# B&R Automation Studio project 8238 (part 21)

#### mnTestCyclic.st - Cyclic code
```iecst
(********************************************************************
 * COPYRIGHT -- Herbert Kannegiesser GmbH
 ********************************************************************
 * Program: mnTest
 * File: mnTestCyclic.st
 * Author: hunholz
 * Created: March 03, 2012
 ********************************************************************
 * Implementation of program mnTest
 ********************************************************************)

PROGRAM _CYCLIC

	//====================
	// Kommandointerpreter
	//====================

	CASE _CommandoState OF

		_csIdle:

			CASE mnTestCmd.Request.Command.wCommand OF

				KG_CMD_NOCOMMAND:

					mnTestCmd.Response.wCmdStatus := KG_CMD_NOCOMMAND;

				MNTEST_CMD_RESET:

					IF mnTestCmd.Request.Command.lData0 <> MNTEST_RESETMODE_WARMSTART AND mnTestCmd.Request.Command.lData0 <> MNTEST_RESETMODE_COLDSTART THEN

						mnTestCmd.Response.wCmdStatus := KG_CMDSTAT_INVALID_PARAMETER;

					ELSE

						SYSreset(enable := TRUE, mode := UDINT_TO_USINT(mnTestCmd.Request.Command.lData0));
						mnTestCmd.Response.wCmdStatus := MNTEST_CMD_RESET;

					END_IF

					_CommandoState := _csWaitForNull;

				MNTEST_CMD_SETMODE:

					IF _wTestMode <> 0 THEN

						mnTestCmd.Response.wCmdStatus := MNTEST_CMDSTAT_SETMODEFAILED;

					ELSIF mnTestCmd.Request.Command.lData0 = 0 OR mnTestCmd.Request.Command.lData0 > MNTEST_TESTMODE_MAX THEN

						mnTestCmd.Response.wCmdStatus := KG_CMDSTAT_INVALID_PARAMETER;

					ELSE

						IF IFmnParam.Out.xParamOK THEN
							_wTestMode := UDINT_TO_UINT(mnTestCmd.Request.Command.lData0);
							mnTestCmd.Response.wCmdStatus := MNTEST_CMD_SETMODE;
							_TestState := _tsSetMode;
						END_IF

					END_IF

					_CommandoState := _csWaitForNull;

				ELSE

					_CommandoState := _csWaitForNull;
					mnTestCmd.Response.wCmdStatus := KG_CMDSTAT_NOTVALID;

			END_CASE

		_csWaitForNull:

			IF mnTestCmd.Request.Command.wCommand = KG_CMD_NOCOMMAND THEN

				_CommandoState := _csIdle;
				mnTestCmd.Response.wCmdStatus := KG_CMD_NOCOMMAND;

			END_IF

		ELSE

			_CommandoState := _csIdle;

	END_CASE

	//======================
	// Statemachine Testmode
	//======================

	CASE _TestState OF

		_tsIdle:

			// Tue nichts

		_tsSetMode:

			_sMachineNo := WSTRING_TO_STRING(IFmnParam.Out.utfMachineNumber);

			_fbSetMode(enable := TRUE, pStruc := IFmnTest.In.pStrucTest, wMode := _wTestMode, sMachineNo := _sMachineNo);

			IF _fbSetMode.status = ERR_OK THEN

				IF _wTestMode = 1 THEN

					// Framework darf keine Meldungen mehr erzeugen und das
					// Meldesystem wird zurückgesetzt
					IFmnTest.Out.xNoMessages := TRUE;
					brsmemset(ADR(kgMsgStatus),0,SIZEOF(kgMsgStatus));

					_TestState := _tsPrepTest1;

				ELSIF _wTestMode = 2 THEN

					brsmemset(ADR(kgMsgStatus),0,SIZEOF(kgMsgStatus));

					_TestState := _tsRun;

				END_IF

			ELSE

				_TestState := _tsFault;

				mnTestStat.wStatus := MNTEST_STAT_ERRFBSETMODE;
				mnTestStat.sStatus := UINT_TO_STRING(_fbSetMode.status);

			END_IF

		_tsPrepTest1:

			_doInfoCfg.enable := TRUE;	// VAR_INPUT BOOL enable 'enables execution'
			_doInfoCfg.pName := ADR('CfgMsgStat');	// VAR_INPUT UDINT pName 'name of data object'
			_doInfoCfg();

			IF _doInfoCfg.status = ERR_OK THEN

				_wMsgCnt := UDINT_TO_UINT((_doInfoCfg.len-SIZEOF(UINT))/SIZEOF (MsgCfgLine_Typ)); // Laenge der Version zu Beginn abziehen

				IF _wMsgCnt > 0 AND _wMsgCnt <= MNMSG_MAX_CFGMESSAGES THEN

					_MsgCfgList ACCESS _doInfoCfg.pDatObjMem + SIZEOF(UINT);
					_TestState := _tsRun;

				ELSE
					// Meldungskonfiguration fehlerhaft
					_TestState := _tsFault;

					mnTestStat.wStatus := MNTEST_STAT_ERRMSGCFGCNT;
					mnTestStat.sStatus := UINT_TO_STRING(_wMsgCnt);

				END_IF

			ELSE
				// Meldungskonfiguration fehlt
				_TestState := _tsFault;
				mnTestStat.wStatus := MNTEST_STAT_ERRMSGCFG;
				mnTestStat.sStatus := UINT_TO_STRING(_doInfoCfg.status);

			END_IF

		_tsRun:

			_fbRunTest(enable := TRUE, pStruc := IFmnTest.In.pStrucTest, wMode := _wTestMode, sMachineNo := _sMachineNo);

			IF _fbRunTest.status = KG_ERR_NULPOINTER THEN

				_TestState := _tsFault;

				mnTestStat.wStatus := MNTEST_STAT_FBRUNTEST;
				mnTestStat.sStatus := UINT_TO_STRING(_fbRunTest.status);

			END_IF

			// ACTION RUN MessageTest

			IF _wTestMode = 1 THEN
				_MessageTest1;
			END_IF

		_tsFault:

			// Tue erstmal nichts

	END_CASE

	mnTestStatAd.wMode := _wTestMode;

END_PROGRAM
```

#### mnTestInit.st - Initialization code
```iecst
(********************************************************************
 * COPYRIGHT -- Herbert Kannegiesser GmbH
 ********************************************************************
 * Program: mnTest
 * File: mnTestInit.st
 * Author: hunholz
 * Created: March 03, 2012
 ********************************************************************
 * Implementation of program mnTest
 ********************************************************************)

PROGRAM _INIT

	// Packet-Version auslesen mit MO_ver aus SYS_lib und für den Additional Status zur Verfügung stellen

	_sPkgName := 'mnTestFW';

	IF ( MO_ver(ADR(_sPkgName), 0, ADR(_VerStruc)) = 0 ) THEN

		brsmemcpy(ADR(mnTestStatAd.sPkgVersion), ADR(_VerStruc.version), SIZEOF(_VerStruc.version));

	ELSE

		mnTestStatAd.sPkgVersion := '---';

	END_IF

	// Test ist auf jeden Fall deaktiviert

	_wTestMode := 0;

END_PROGRAM
```

#### mnTestExit.st - Exit code
```iecst
(********************************************************************
 * COPYRIGHT -- Herbert Kannegiesser GmbH
 ********************************************************************
 * Program: mnTest
 * File: mnTestExit.st
 * Author: hunholz
 * Created: March 03, 2012
 ********************************************************************
 * Implementation of program mnTest
 ********************************************************************)

PROGRAM _EXIT

(* TODO : Add your code here *)

END_PROGRAM
```

#### mnTest.typ - Local data types
```iecst
(********************************************************************
 * COPYRIGHT -- Herbert Kannegiesser GmbH
 ********************************************************************
 * Program: mnTest
 * File: mnTest.typ
 * Author: hunholz
 * Created: March 03, 2012
 ********************************************************************
 * Local data types of program mnTest
 ********************************************************************)

TYPE
	_CommandoState_enum :
		(
		_csIdle,
		_csSetTestMode,
		_csWaitForNull
		);
	_TestState_enum :
		(
		_tsIdle,
		_tsSetMode,
		_tsPrepTest1,
		_tsRun,
		_tsFault
		);
END_TYPE
```

#### mnTest.var - Local variables
```iecst
(********************************************************************
 * COPYRIGHT -- Herbert Kannegiesser GmbH
 ********************************************************************
 * Program: mnTest
 * File: mnTest.var
 * Author: hunholz
 * Created: March 03, 2012
 ********************************************************************
 * Local variables of program mnTest
 ********************************************************************)
(*Packageversion auslesen*)
VAR
	_sPkgName : STRING[10];
	_VerStruc : MoVerStruc_typ;
END_VAR
(*Aktueller Testmodus*)
VAR
	_wTestMode : UINT := 0;
END_VAR
(*Kommandointerpreter*)
VAR
	_CommandoState : _CommandoState_enum;
	_TestState : _TestState_enum;
	_fbSetMode : TestUser_SetMode;
	_fbRunTest : TestUser_RunTest;
	_doInfoCfg : DatObjInfo;
	_wMsgCnt : UINT;
	_MsgCfgList : REFERENCE TO ARRAY[1..MNMSG_MAX_CFGMESSAGES] OF MsgCfgLine_Typ;
	_ii : UINT;
END_VAR
VAR CONSTANT
	_MNTEST_MAX_MSGGROUPS : UINT := 30;
END_VAR
VAR
	_TONmsgclk2 : TON;
	_TONmsgclk1 : TON;
	_wMsgTick : UINT;
	_wStateMsgTest : ARRAY[1.._MNTEST_MAX_MSGGROUPS] OF UINT;
	_xReason : ARRAY[1.._MNTEST_MAX_MSGGROUPS] OF BOOL;
	_wMsgIdxOffset : ARRAY[1.._MNTEST_MAX_MSGGROUPS] OF UINT;
	_wMsgClass : ARRAY[0..4] OF UINT := [0,1,10,11,20];
	_TONMsg : ARRAY[1.._MNTEST_MAX_MSGGROUPS] OF TON;
	_TONMsgPause : ARRAY[1.._MNTEST_MAX_MSGGROUPS] OF TON;
	_sMachineNo : STRING[15];
	_tMsgGap : TIME := T#10s;
	_lGap : UDINT;
END_VAR
```

#### _MessageTest1.st
```iecst
(********************************************************************
 * COPYRIGHT -- Herbert Kannegiesser GmbH
 ********************************************************************
 * Program: mnTest
 * File: _MessageTest1.st
 * Author: hunholz
 * Created: March 07, 2012
 ********************************************************************
 * Implementation of program mnTest
 ********************************************************************)

(* Meldungen zyklisch bearbeiten *)
ACTION _MessageTest1:

	_TONmsgclk1(IN := NOT _TONmsgclk2.Q, PT := _tMsgGap);
	_TONmsgclk2(IN := _TONmsgclk1.Q, PT := T#100ms);

	// Bug 781 : Meldungsabstände in der Simulation sporadisch verkürzen

	IF EDGEPOS(_TONmsgclk1.Q) THEN
		_wMsgTick := _wMsgTick + 1;
		_lGap := DINT_TO_UDINT( ((ABS(IFmnSystem.In.PLC.diSystemTime) / 100000 / 3) MOD 100) * 100);
		_tMsgGap := UDINT_TO_TIME(_lGap);
	END_IF

	IF _wMsgTick > _MNTEST_MAX_MSGGROUPS THEN
		_wMsgTick := 1;
	END_IF

	FOR _ii := 1 TO _MNTEST_MAX_MSGGROUPS DO

		CASE _wStateMsgTest[_ii] OF

			0:
				IF (_ii + _wMsgIdxOffset[_ii]) <= _wMsgCnt THEN
					// Warte auf Meldungsbeginn
					IF _ii = _wMsgTick THEN
						// Meldung setzen
						_xReason[_ii] := TRUE;
						kgMsgStatus[_ii].wFunction_ID := _MsgCfgList[_ii+_wMsgIdxOffset[_ii]].wFunction_ID;
						kgMsgStatus[_ii].wInstance := _MsgCfgList[_ii+_wMsgIdxOffset[_ii]].wInstance;

						IF _wMsgClass[_ii MOD 5] = MNMSG_CLASS_MAINTENANCE THEN
							kgMsgStatus[_ii].diMaintAttr1 := _ii;
							kgMsgStatus[_ii].diMaintAttr2 := _ii + 100;
							kgMsgStatus[_ii].sMaintAttrTxt := UINT_TO_STRING(_ii);
							kgMsgStatus[_ii].wMaintAckLevel := MNMSG_CLASS_NO_ACK;
							kgMsgStatus[_ii].wMaintNumber := _MsgCfgList[_ii+_wMsgIdxOffset[_ii]].wMsgNumber;
							kgMsgStatus[_ii].wMsgClass := MNMSG_CLASS_MAINTENANCE;
						ELSE
							kgMsgStatus[_ii].diMsgAttr1 := _ii;
							kgMsgStatus[_ii].diMsgAttr2 := _ii + 100;
							kgMsgStatus[_ii].sMsgAttrTxt := UINT_TO_STRING(_ii);
							kgMsgStatus[_ii].wMsgAckLevel := SEL((_wMsgClass[_ii MOD 4] < 10),0,MNMSG_CLASS_NO_ACK);
							kgMsgStatus[_ii].wMsgNumber := _MsgCfgList[_ii+_wMsgIdxOffset[_ii]].wMsgNumber;
							kgMsgStatus[_ii].wMsgClass := _wMsgClass[_ii MOD 5];
						END_IF

						_wStateMsgTest[_ii] := 1;

					END_IF
				ELSE
					_wMsgIdxOffset[_ii] := 0;
				END_IF

			1:
				// Warte bis Meldung beendet
				IF _TONMsg[_ii].Q THEN

					_xReason[_ii] := FALSE;

					IF kgMsgStatus[_ii].wMaintAckLevel = MNMSG_CLASS_NO_ACK THEN

						kgMsgStatus[_ii].wMaintAckLevel := _ii MOD 4;
						_wStateMsgTest[_ii] := 10;

					ELSIF kgMsgStatus[_ii].wMsgAckLevel = MNMSG_CLASS_NO_ACK THEN

						kgMsgStatus[_ii].wMsgAckLevel := _ii MOD 4;
						_wStateMsgTest[_ii] := 20;

					ELSE

						_wStateMsgTest[_ii] := 99;

					END_IF

				END_IF

			10:
			// Warten auf Wartungsquittierung

				IF kgMsgStatus[_ii].xAckMaint THEN
					kgMsgStatus[_ii].xAckRead := TRUE;
					_wStateMsgTest[_ii] := 99;
				END_IF

			20:
				// Warten auf Störungsquittierung

				IF kgMsgStatus[_ii].xAckFault THEN
					kgMsgStatus[_ii].xAckRead := TRUE;
					_wStateMsgTest[_ii] := 99;
				END_IF

			99:
				// Meldung entfernen
				kgMsgStatus[_ii].diMaintAttr1 := 0;
				kgMsgStatus[_ii].diMaintAttr2 := 0;
				kgMsgStatus[_ii].sMaintAttrTxt := '';
				kgMsgStatus[_ii].wMaintAckLevel := 0;
				kgMsgStatus[_ii].wMaintNumber := 0;
				kgMsgStatus[_ii].xAckRead := FALSE;
				kgMsgStatus[_ii].wMsgClass := 0;
				kgMsgStatus[_ii].diMsgAttr1 := 0;
				kgMsgStatus[_ii].diMsgAttr2 := 0;
				kgMsgStatus[_ii].sMsgAttrTxt := '';
				kgMsgStatus[_ii].wMsgAckLevel := 0;
				kgMsgStatus[_ii].wMsgNumber := 0;
				kgMsgStatus[_ii].wFunction_ID := 0;
				kgMsgStatus[_ii].wInstance := 0;

				_wStateMsgTest[_ii] := 100;

			100:
				// Warten bis Wartezeit beendet
				IF _TONMsgPause[_ii].Q THEN
					_wMsgIdxOffset[_ii] := _wMsgIdxOffset[_ii] + _MNTEST_MAX_MSGGROUPS;
					_wStateMsgTest[_ii] := 0;
				END_IF

		END_CASE

		_TONMsg[_ii](IN := _xReason[_ii], PT := T#10m);
		_TONMsgPause[_ii](IN := NOT _xReason[_ii], PT := T#4m);

	END_FOR

END_ACTION
```

### Package Logical/Standard/Kanlink/KGFramework/Pkg_svCPCache - Category-Program-Verwaltung

### Pkg_svCPCache.typ - Global data types
```iecst
(********************************************************************
 * COPYRIGHT -- Herbert Kannegiesser GmbH
 ********************************************************************
 * Package: Pkg_svCPCache
 * File: Pkg_svCPCache.typ
 * Author: hunholz
 * Created: March 29, 2012
 ********************************************************************
 * Data types of package Pkg_svCPCache
 ********************************************************************)

TYPE
	svCPCache_Relation_Typ : 	STRUCT
		dtTimestamp : DATE_AND_TIME;
		sCategory : STRING[11];
		wProgramNo : UINT;
	END_STRUCT;
	IFsvCPCache_In_Typ : 	STRUCT
		wCmd : UINT;
		wReqUseDB : UINT;
		sReqCategory : STRING[11];
		utfReqCategoryName : WSTRING[31];
		wReqProgramNo : UINT;
		wReqLoadrate : UINT;
		rReqSoilfactor : REAL;
		wReqColidxFor : UINT;
		wReqColidxBack : UINT;
		wSetOffset : UINT;
		sImpDevice : STRING[31];
		sImpPath : STRING[31];
	END_STRUCT;
	IFsvCPCache_Out_Typ : 	STRUCT
		xReady : BOOL;
		xListReady : BOOL;
		wCmdResponse : UINT;
		wCntRelations : UINT;
		wRespFromDB : UINT;
		utfRespCategoryName : WSTRING[31];
		rRespSoilFactor : REAL;
		wRespColidxFor : UINT;
		wRespColidxBack : UINT;
		wRespLoadrate : UINT;
		wRespProgramNo : UINT;
		utfRespProgramName : WSTRING[31];
		wListOffset : UINT;
		wListCnt : UINT;
		sListCategory : ARRAY[1..SVCPCACHE_CNT_LISTRELATIONS]OF STRING[11];
		utfListCategoryname : ARRAY[1..SVCPCACHE_CNT_LISTRELATIONS]OF WSTRING[31];
		wListProgramNo : ARRAY[1..SVCPCACHE_CNT_LISTRELATIONS]OF UINT;
		utfListProgramName : ARRAY[1..SVCPCACHE_CNT_LISTRELATIONS]OF WSTRING[31];
	END_STRUCT;
	IFsvCPCache_Typ : 	STRUCT
		In : IFsvCPCache_In_Typ;
		Out : IFsvCPCache_Out_Typ;
	END_STRUCT;
	svCPCacheStatAd_Typ : 	STRUCT
		xReady : BOOL;
		sPkgVersion : STRING[10];
	END_STRUCT;
END_TYPE
```

### Pkg_svCPCache.var - Global variables
```iecst
(********************************************************************
 * COPYRIGHT -- Herbert Kannegiesser GmbH
 ********************************************************************
 * Package: Pkg_svCPCache
 * File: Pkg_svCPCache.var
 * Author: hunholz
 * Created: March 29, 2012
 ********************************************************************
 * Variables of package Pkg_svCPCache
 ********************************************************************)
(*KONSTANTEN*)
VAR CONSTANT
	SVCPCACHE_DBREQ_LOCAL : UINT := 0;
	SVCPCACHE_DBREQ_DFII : UINT := 1;
END_VAR
(*Kommandos*)
VAR CONSTANT
	SVCPCACHE_CMD_GETPROG : UINT := 1;
	SVCPCACHE_CMD_INSERTCATEGORY : UINT := 2;
	SVCPCACHE_CMD_UPDATECATEGORY : UINT := 3;
	SVCPCACHE_CMD_DELETECATEGORY : UINT := 4;
	SVCPCACHE_CMD_SETOFFSET : UINT := 5;
	SVCPCACHE_CMD_RESTORE : UINT := 6;
END_VAR
(*Status*)
VAR CONSTANT
	SVCPCACHE_STAT_MEMALLOC : UINT := 60000;
	SVCPCACHE_STAT_CREATEFILE : UINT := 60001;
	SVCPCACHE_STAT_WRITEFILE : UINT := 60002;
	SVCPCACHE_STAT_OPENFILE : UINT := 60003;
	SVCPCACHE_STAT_NOSPACE : UINT := 60004;
	SVCPCACHE_STAT_INVALIDCATEGORY : UINT := 60005;
	SVCPCACHE_STAT_CATEGORYEXIST : UINT := 60006;
	SVCPCACHE_STAT_CATEGORYNOTEXIST : UINT := 60007;
	SVCPCACHE_STAT_CATEGORYLISTEMPTY : UINT := 60008;
	SVCPCACHE_STAT_DBNOTREADY : UINT := 60009;
	SVCPCACHE_STAT_FILENOTFOUND : UINT := 60010;
END_VAR
(*Schnittstellen*)
VAR
	IFsvCPCache : IFsvCPCache_Typ;
	svCPCacheStatAd : svCPCacheStatAd_Typ;
END_VAR
```

### Program Logical/Standard/Kanlink/KGFramework/Pkg_svCPCache/svCPCache (IEC) - Category-Program-Cache

#### svCPCacheCyclic.st - Cyclic code
```iecst
(********************************************************************
 * COPYRIGHT -- Herbert Kannegiesser GmbH
 ********************************************************************
 * Program: svCPCache
 * File: svCPCacheCyclic.st
 * Author: hunholz
 * Created: March 29, 2012
 ********************************************************************
 * Implementation of program svCPCache
 ********************************************************************)

PROGRAM _CYCLIC

	// Zyklische Arbeit. Entgegennehmen von Aufträgen
	IF _xCacheReady THEN

		// Kommandos abarbeiten
		_actIFCmd;

		// CSV-File speichern
		_actSaveCSV;

	END_IF

	// Erstmaliges Lesen der Kategorie-Programm-Zuordnung
	IF _xCacheInitReady AND NOT _xCacheReady AND IFmnParam.Out.xParamOK THEN

		_sDevice := KG_DEVICE_COMPACTFLASH;
		_sPathFile := CONCAT(_SVCPCACHE_CSV_PATH, _SVCPCACHE_CSV_FILE);

		IF _enImport = cs_ImpIdle THEN
			_enImport := cs_ImpStart;
		END_IF

		///////////////////////////////
		// ACTION
		///////////////////////////////
		_actCPImport;

		IF _enImport = cs_ImpRdyFault THEN

			// Einlesen mit Fehler abgebrochen
			_xCacheInitReady := FALSE;

			_enImport := cs_ImpIdle;

		ELSIF _enImport = cs_ImpRdySuccess THEN

			// Erfolgreich eingelesen
			_xCacheReady := TRUE;

			IFsvCPCache.Out.xListReady := TRUE;
			IFsvCPCache.Out.wCntRelations := _wCntRelations;

			// Liste füllen
			IFsvCPCache.Out.wListOffset := 0;
			_actFillCPList;

			_enImport := cs_ImpIdle;

		END_IF

	END_IF

	IFsvCPCache.Out.xReady := _xCacheReady;
	svCPCacheStatAd.xReady := _xCacheReady;

END_PROGRAM
```

#### svCPCacheInit.st - Initialization code
```iecst
(********************************************************************
 * COPYRIGHT -- Herbert Kannegiesser GmbH
 ********************************************************************
 * Program: svCPCache
 * File: svCPCacheInit.st
 * Author: hunholz
 * Created: March 29, 2012
 ********************************************************************
 * Implementation of program svCPCache
 ********************************************************************)

PROGRAM _INIT

	// Packet-Version auslesen mit MO_ver aus SYS_lib und für den Additional Status zur Verfügung stellen

	_sPkgName := 'svCPCache';

	IF ( MO_ver(ADR(_sPkgName), 0, ADR(_VerStruc)) = 0 ) THEN

		brsmemcpy(ADR(svCPCacheStatAd.sPkgVersion), ADR(_VerStruc.version), SIZEOF(_VerStruc.version));

	ELSE

		svCPCacheStatAd.sPkgVersion := '---';

	END_IF

	_xCacheInitReady := FALSE;

	REPEAT // UNTIL TRUE

		// Schleife, die nur einmal durchlaufen wird, aber jederzeit verlassen werden kann
		#pragma warning ( disable : 1288 )
		//Mögliche Optionen
		//SVCPCACHE_DBREQ_NO = 0
		//SVCPCACHE_DBREQ_DFII = 1
		IF SVCPCACHE_DB_REQUEST > 1 THEN
			EXIT;
		END_IF

		#pragma warning ( default : 1288 )

		//Container sind von 0..20 möglich
		IF SVCPCACHE_NO_INDCONTAINER > 20 THEN
			EXIT;
		END_IF

		// Speicher zum Parsen und Schreiben allokieren

		_lMemLen := SVCPCACHE_CNT_RELATIONS * 146 + 200;

		_MemPartCreate(enable := TRUE, len := _lMemLen + 100);

		IF _MemPartCreate.status <> ERR_OK THEN
			EXIT;
		END_IF

		_xCacheInitReady := TRUE;

		UNTIL TRUE

	END_REPEAT

END_PROGRAM
```

#### svCPCacheExit.st - Exit code
```iecst
(********************************************************************
 * COPYRIGHT -- Herbert Kannegiesser GmbH
 ********************************************************************
 * Program: svCPCache
 * File: svCPCacheExit.st
 * Author: hunholz
 * Created: March 29, 2012
 ********************************************************************
 * Implementation of program svCPCache
 ********************************************************************)

PROGRAM _EXIT

(* TODO : Add your code here *)

END_PROGRAM
```

#### svCPCache.typ - Local data types
```iecst
(********************************************************************
 * COPYRIGHT -- Herbert Kannegiesser GmbH
 ********************************************************************
 * Program: svCPCache
 * File: svCPCache.typ
 * Author: hunholz
 * Created: March 29, 2012
 ********************************************************************
 * Local data types of program svCPCache
 ********************************************************************)

TYPE
	enum_CmdCP :
		(
		cs_CmdIdle,
		cs_CmdSave,
		cs_CmdWaitForDB,
		cs_CmdImport,
		cs_CmdWaitForNoCommand
		);
	enum_ImportCP :
		(
		cs_ImpIdle,
		cs_ImpStart,
		cs_ImpFileOpen,
		cs_ImpFileRead,
		cs_ImpFileClose,
		cs_ImpParse,
		cs_ImpRdySuccess,
		cs_ImpRdyFault
		);
	enum_SaveCP :
		(
		cs_SaveIdle,
		cs_SaveCreateCSV,
		cs_SaveDeleteFile,
		cs_SaveCreateFile,
		cs_SaveOpenFile,
		cs_SaveWriteFile,
		cs_SaveCloseFile,
		cs_SaveRdySuccess,
		cs_SaveRdyFault
		);
END_TYPE
```

#### svCPCache.var - Local variables
```iecst
(********************************************************************
 * COPYRIGHT -- Herbert Kannegiesser GmbH
 ********************************************************************
 * Program: svCPCache
 * File: svCPCache.var
 * Author: hunholz
 * Created: March 29, 2012
 ********************************************************************
 * Local variables of program svCPCache
 ********************************************************************)
VAR CONSTANT
	_SVCPCACHE_CSV_FILE : STRING[15] := 'cpcache.csv';
	_SVCPCACHE_CSV_PATH : STRING[31] := 'PM\Export\';
END_VAR
VAR
	_sPkgName : STRING[11];
	_VerStruc : MoVerStruc_typ;
	_CPCache : ARRAY[1..SVCPCACHE_CNT_RELATIONS] OF mnParam_CProw_typ;
	_wCntRelations : UINT;
	_i : UINT;
	_lMemLen : UDINT;
	_lLineAdress : ARRAY[1..SVCPCACHE_MAX_PARSELINES] OF UDINT;
	_wLineLen : ARRAY[1..SVCPCACHE_MAX_PARSELINES] OF UINT;
	_wStartLine : UINT;
	_CountLines : mnParam_CountLines;
	_GetCsvDat : mnParam_GetCsvDat;
	_enCmd : enum_CmdCP;
	_enImport : enum_ImportCP;
	_enSave : enum_SaveCP;
	_xImpFault : BOOL;
	_xImpReady : BOOL;
	_MemPartCreate : AsMemPartCreate;
	_FileOpen : FileOpen;
	_FileRead : FileRead;
	_FileClose : FileClose;
	_MemPartAllocClear : AsMemPartAllocClear;
	_MemPartFree : AsMemPartFree;
	_lTempMem : UDINT;
	_lFileLen : UDINT;
	_xCacheInitReady : BOOL;
	_xCacheReady : BOOL;
	_wfcli : UINT;
	_wfclj : UINT;
	_SaveMemPartAlloc : AsMemPartAllocClear;
	_lWriteSize : UDINT;
	_WriteBOM : mnParam_WriteBOM_Mem;
	_WriteComment : mnParam_WriteCSV254_Mem;
	_WriteNewLine : mnParam_WriteNewline_Mem;
	_MachineNoRow : mnParam_HeaderMachineNoRow_typ;
	_WriteMachineNo : mnParam_WriteCSV252_Mem;
	_DTGetTime : DTGetTime;
	_HeaderTimeRow : mnParam_HeaderTimeRow_typ;
	_WriteTimeStamp : mnParam_WriteCSV251_Mem;
	_sci : UINT;
	_WriteCP : mnParam_WriteCSV81_Mem;
	_FileCreate : FileCreate;
	_FileDelete : FileDelete;
	_wSaveCSVstatus : UINT;
	_SaveMemPartFree : AsMemPartFree;
	_FileWrite : FileWrite;
	_sCategory : STRING[11];
	_xCategoryExist : BOOL;
	_wCmd : UINT;
	_TrimCat : _TrimCategory;
	_wCategoryIdx : UINT;
	_sDevice : STRING[31];
	_sPathFile : STRING[31];
END_VAR
```

#### _actCPImport.st
```iecst
(********************************************************************
 * COPYRIGHT -- Herbert Kannegiesser GmbH
 ********************************************************************
 * Program: svCPCache
 * File: _actCPImport.st
 * Author: hunholz
 * Created: March 29, 2012
 ********************************************************************
 * Implementation of program svCPCache
 ********************************************************************)

(* Kategorie-Programm-Zuordnung aus CSV-Datei lesen *)
ACTION _actCPImport:

	CASE _enImport OF

		cs_ImpIdle:

			// Tue nichts

		cs_ImpStart:

			// Initialisierung
			brsmemset(ADR(_CPCache), 0, SIZEOF(_CPCache));
			brsmemset(ADR(_lLineAdress), 0, SIZEOF(_lLineAdress));
			brsmemset(ADR(_wLineLen), 0, SIZEOF(_wLineLen));
			_wCntRelations := 0;
			_xImpFault := FALSE;
			_xImpReady := FALSE;
			_lTempMem := 0;

			_enImport := cs_ImpFileOpen;

		cs_ImpFileOpen:

			_FileOpen(enable := TRUE, pDevice := ADR(_sDevice), pFile := ADR(_sPathFile), mode := fiREAD_ONLY);

			IF _FileOpen.status = ERR_OK THEN

				IF _FileOpen.filelen > SIZEOF(KGBOM) THEN

					_lFileLen := _FileOpen.filelen - SIZEOF(KGBOM);

					_MemPartAllocClear(enable := TRUE, ident := _MemPartCreate.ident, len := _lFileLen);

					IF _MemPartAllocClear.status = ERR_OK THEN

						_lTempMem := _MemPartAllocClear.mem;
						_enImport := cs_ImpFileRead;

					ELSE

						_xImpFault := TRUE;
						_enImport := cs_ImpFileClose;

					END_IF

				ELSE

					_xImpReady := TRUE;
					_enImport := cs_ImpFileClose;

				END_IF

			ELSIF _FileOpen.status <> ERR_FUB_BUSY THEN

				_enImport := cs_ImpRdySuccess;

			END_IF

		cs_ImpFileRead:

			_FileRead(enable := TRUE, ident := _FileOpen.ident, offset := SIZEOF(KGBOM), pDest := _MemPartAllocClear.mem, len := _lFileLen);

			IF _FileRead.status <> ERR_FUB_BUSY THEN

				IF _FileRead.status <> ERR_OK THEN

					_xImpFault := TRUE;

				END_IF

				_enImport := cs_ImpFileClose;

			END_IF

		cs_ImpFileClose:

			_FileClose(enable := TRUE, ident := _FileOpen.ident);

			IF _FileClose.status = ERR_OK THEN

				IF _xImpFault THEN

					_enImport := cs_ImpRdyFault;

					IF _lTempMem <> 0 THEN
						_MemPartFree(enable := TRUE, ident := _MemPartAllocClear.ident, mem := _lTempMem);
					END_IF

				ELSIF _xImpReady THEN

					_enImport := cs_ImpRdySuccess;

					IF _lTempMem <> 0 THEN
						_MemPartFree(enable := TRUE, ident := _MemPartAllocClear.ident, mem := _lTempMem);
					END_IF

				ELSE

					_enImport := cs_ImpParse;

				END_IF

			ELSIF _FileClose.status <> ERR_FUB_BUSY THEN

				_enImport := cs_ImpRdyFault;

			END_IF

		cs_ImpParse:

			_CountLines.enable 	:= TRUE;
			_CountLines.pFile 		:= _lTempMem;
			_CountLines.FileSize 	:= _lFileLen;
			_CountLines.MaxLines	:= SVCPCACHE_MAX_PARSELINES;
			_CountLines.pAdresses	:= ADR(_lLineAdress);
			_CountLines.pLens		:= ADR(_wLineLen);

			_CountLines();

			IF _CountLines.status <> ERR_OK THEN

				_MemPartFree(enable := TRUE, ident := _MemPartAllocClear.ident, mem := _lTempMem);
				_enImport := cs_ImpRdyFault;

			ELSE

				_wStartLine := 1;

				REPEAT

					_GetCsvDat.enable := TRUE;
					brwcsncpy( ADR(_GetCsvDat.utfCsvString), _lLineAdress[_wStartLine], MIN(299, _wLineLen[_wStartLine]));
					_GetCsvDat();

					IF _GetCsvDat.RowType = MNPARAM_CSV_CP AND _wCntRelations < SVCPCACHE_CNT_RELATIONS THEN

						_wCntRelations := _wCntRelations + 1;

						_CPCache[_wCntRelations] := _GetCsvDat.CsvCProw;

					END_IF

					_wStartLine := _wStartLine + 1;

					UNTIL
					_wStartLine > _CountLines.CntLines

				END_REPEAT

				_MemPartFree(enable := TRUE, ident := _MemPartAllocClear.ident, mem := _lTempMem);
				_enImport := cs_ImpRdySuccess;

			END_IF

		cs_ImpRdySuccess:

			// Beendet mit Erfolg

		cs_ImpRdyFault:

			// Mit Fehler beendet

	END_CASE

END_ACTION
```

#### _actIFCmd.st
```iecst
(********************************************************************
 * COPYRIGHT -- Herbert Kannegiesser GmbH
 ********************************************************************
 * Program: svCPCache
 * File: _actIFCmd.st
 * Author: hunholz
 * Created: March 30, 2012
 ********************************************************************
 * Implementation of program svCPCache
 ********************************************************************)

(* Add a new action to your IEC program or library *)
ACTION _actIFCmd:

	CASE _enCmd OF

		cs_CmdIdle:

		// Warte auf Kommando

			CASE IFsvCPCache.In.wCmd OF

				KG_CMD_NOCOMMAND:

					IFsvCPCache.Out.wCmdResponse := KG_CMD_NOCOMMAND;

				SVCPCACHE_CMD_GETPROG:

					IFsvCPCache.Out.rRespSoilFactor 		:= 1.0;
					IFsvCPCache.Out.utfRespCategoryName		:= "";
					IFsvCPCache.Out.wRespColidxBack			:= 15;
					IFsvCPCache.Out.wRespColidxFor			:= 1;
					IFsvCPCache.Out.wRespLoadrate			:= 100;
					IFsvCPCache.Out.wRespProgramNo			:= 0;
					IFsvCPCache.Out.utfRespProgramName		:= "";

					IFsvCPCache.Out.wRespFromDB				:= SVCPCACHE_DBREQ_LOCAL;

					_TrimCat(sCategory := IFsvCPCache.In.sReqCategory);
					_sCategory := _TrimCat.sOutCategory;

					IF _sCategory <> '' THEN

						// Suche Kategorie auf jeden Fall lokal

						_xCategoryExist := FALSE;
						_wCategoryIdx := 0;

						FOR _i := 1 TO SVCPCACHE_CNT_RELATIONS DO

							IF _CPCache[_i].dtTimeStamp = USINT_TO_DT(0) THEN
								EXIT;
							ELSIF _CPCache[_i].sCategory = _sCategory THEN
								_xCategoryExist := TRUE;
								_wCategoryIdx := _i;
								EXIT;
							END_IF

						END_FOR

						// Entscheidung, ob in der Datenbank gesucht werden soll

						IF IFsvCPCache.In.wReqUseDB = SVCPCACHE_DBREQ_LOCAL THEN

							IF _xCategoryExist THEN

								IFsvCPCache.Out.rRespSoilFactor 		:= _CPCache[_wCategoryIdx].rSoilfactor;
								IFsvCPCache.Out.utfRespCategoryName		:= _CPCache[_wCategoryIdx].utfCategoryName;
								IFsvCPCache.Out.wRespColidxBack			:= _CPCache[_wCategoryIdx].wColBack;
								IFsvCPCache.Out.wRespColidxFor			:= _CPCache[_wCategoryIdx].wColFor;
								IFsvCPCache.Out.wRespLoadrate			:= _CPCache[_wCategoryIdx].wLoadrate;
								IFsvCPCache.Out.wRespProgramNo			:= _CPCache[_wCategoryIdx].wProgramNo;

								FOR _i := 1 TO IFmnParam.Out.Edit.wCntNamelist DO

									IF IFmnParam.Out.Edit.wNameListNo[_i] = IFsvCPCache.Out.wRespProgramNo THEN
										IFsvCPCache.Out.utfRespProgramName := IFmnParam.Out.Edit.utfNameListName[_i];
										EXIT;
									END_IF

								END_FOR

								IFsvCPCache.Out.wCmdResponse := SVCPCACHE_CMD_GETPROG;
								_enCmd := cs_CmdWaitForNoCommand;

							ELSE

								IFsvCPCache.Out.wCmdResponse := SVCPCACHE_STAT_CATEGORYNOTEXIST;
								_enCmd := cs_CmdWaitForNoCommand;

							END_IF

						ELSE // Abfrage der Datenbank starten

							IF IFhlDFII.Out.xConnected THEN

								IFsvCPCache.Out.wCmdResponse := KG_STAT_BUSY;
								_enCmd := cs_CmdWaitForDB;

							ELSE

								IFsvCPCache.Out.wCmdResponse := SVCPCACHE_STAT_DBNOTREADY;
								_enCmd := cs_CmdWaitForNoCommand;

								IF _xCategoryExist THEN

									IFsvCPCache.Out.rRespSoilFactor 		:= _CPCache[_wCategoryIdx].rSoilfactor;
									IFsvCPCache.Out.utfRespCategoryName		:= _CPCache[_wCategoryIdx].utfCategoryName;
									IFsvCPCache.Out.wRespColidxBack			:= _CPCache[_wCategoryIdx].wColBack;
									IFsvCPCache.Out.wRespColidxFor			:= _CPCache[_wCategoryIdx].wColFor;
									IFsvCPCache.Out.wRespLoadrate			:= _CPCache[_wCategoryIdx].wLoadrate;
									IFsvCPCache.Out.wRespProgramNo			:= _CPCache[_wCategoryIdx].wProgramNo;

									FOR _i := 1 TO IFmnParam.Out.Edit.wCntNamelist DO

										IF IFmnParam.Out.Edit.wNameListNo[_i] = IFsvCPCache.Out.wRespProgramNo THEN
											IFsvCPCache.Out.utfRespProgramName := IFmnParam.Out.Edit.utfNameListName[_i];
											EXIT;
										END_IF

									END_FOR

								END_IF

							END_IF

						END_IF

					ELSE

						IFsvCPCache.Out.wCmdResponse := SVCPCACHE_STAT_INVALIDCATEGORY;
						_enCmd := cs_CmdWaitForNoCommand;

					END_IF

				SVCPCACHE_CMD_INSERTCATEGORY:

					_wCmd := SVCPCACHE_CMD_INSERTCATEGORY;

					IF IFsvCPCache.Out.wCntRelations < SVCPCACHE_CNT_RELATIONS THEN

						_TrimCat(sCategory := IFsvCPCache.In.sReqCategory);
						_sCategory := _TrimCat.sOutCategory;

						IF _sCategory <> '' THEN

							_xCategoryExist := FALSE;

							FOR _i := 1 TO SVCPCACHE_CNT_RELATIONS DO

								IF _CPCache[_i].dtTimeStamp = USINT_TO_DT(0) THEN
									EXIT;
								ELSIF _CPCache[_i].sCategory = _sCategory THEN
									_xCategoryExist := TRUE;
									EXIT;
								END_IF

							END_FOR

							IF NOT _xCategoryExist THEN

								_DTGetTime(enable := TRUE);

								FOR _i := 1 TO SVCPCACHE_CNT_RELATIONS DO

									IF _CPCache[_i].dtTimeStamp = USINT_TO_DT(0) THEN

										_CPCache[_i].dtTimeStamp := _DTGetTime.DT1;
										_CPCache[_i].sCategory := _sCategory;
										_CPCache[_i].utfCategoryName := IFsvCPCache.In.utfReqCategoryName;
										_CPCache[_i].wProgramNo := IFsvCPCache.In.wReqProgramNo;
										_CPCache[_i].rSoilfactor := IFsvCPCache.In.rReqSoilfactor;
										_CPCache[_i].wLoadrate := IFsvCPCache.In.wReqLoadrate;
										_CPCache[_i].wColFor := IFsvCPCache.In.wReqColidxFor;
										_CPCache[_i].wColBack := IFsvCPCache.In.wReqColidxBack;

										IFsvCPCache.Out.wCntRelations := IFsvCPCache.Out.wCntRelations + 1;

										EXIT;

									ELSIF brsstrcmp(ADR(_CPCache[_i].sCategory),ADR(_sCategory)) > 0 THEN

										brsmemmove(ADR(_CPCache[_i+1]), ADR(_CPCache[_i]), SIZEOF(_CPCache[1])*(IFsvCPCache.Out.wCntRelations-_i+1) );

										_CPCache[_i].dtTimeStamp := _DTGetTime.DT1;
										_CPCache[_i].sCategory := _sCategory;
										_CPCache[_i].utfCategoryName := IFsvCPCache.In.utfReqCategoryName;
										_CPCache[_i].wProgramNo := IFsvCPCache.In.wReqProgramNo;
										_CPCache[_i].rSoilfactor := IFsvCPCache.In.rReqSoilfactor;
										_CPCache[_i].wLoadrate := IFsvCPCache.In.wReqLoadrate;
										_CPCache[_i].wColFor := IFsvCPCache.In.wReqColidxFor;
										_CPCache[_i].wColBack := IFsvCPCache.In.wReqColidxBack;

										IFsvCPCache.Out.wCntRelations := IFsvCPCache.Out.wCntRelations + 1;

										EXIT;

									END_IF

								END_FOR

								_enSave := cs_SaveCreateCSV;

								_enCmd := cs_CmdSave;

							ELSE

								IFsvCPCache.Out.wCmdResponse := SVCPCACHE_STAT_CATEGORYEXIST;
								_enCmd := cs_CmdWaitForNoCommand;

							END_IF

						ELSE

							IFsvCPCache.Out.wCmdResponse := SVCPCACHE_STAT_INVALIDCATEGORY;
							_enCmd := cs_CmdWaitForNoCommand;

						END_IF

					ELSE

						IFsvCPCache.Out.wCmdResponse := SVCPCACHE_STAT_NOSPACE;
						_enCmd := cs_CmdWaitForNoCommand;

					END_IF

				SVCPCACHE_CMD_UPDATECATEGORY:

					_wCmd := SVCPCACHE_CMD_UPDATECATEGORY;

					IF IFsvCPCache.Out.wCntRelations > 0 THEN

						_TrimCat(sCategory := IFsvCPCache.In.sReqCategory);
						_sCategory := _TrimCat.sOutCategory;

						IF _sCategory <> '' THEN

							_xCategoryExist := FALSE;

							FOR _i := 1 TO SVCPCACHE_CNT_RELATIONS DO

								IF _CPCache[_i].dtTimeStamp = USINT_TO_DT(0) THEN
									EXIT;
								ELSIF _CPCache[_i].sCategory = _sCategory THEN
									_xCategoryExist := TRUE;
									EXIT;
								END_IF

							END_FOR

							IF _xCategoryExist THEN

								_DTGetTime(enable := TRUE);

								_CPCache[_i].dtTimeStamp := _DTGetTime.DT1;
								_CPCache[_i].sCategory := _sCategory;
								_CPCache[_i].utfCategoryName := IFsvCPCache.In.utfReqCategoryName;
								_CPCache[_i].wProgramNo := IFsvCPCache.In.wReqProgramNo;
								_CPCache[_i].rSoilfactor := IFsvCPCache.In.rReqSoilfactor;
								_CPCache[_i].wLoadrate := IFsvCPCache.In.wReqLoadrate;
								_CPCache[_i].wColFor := IFsvCPCache.In.wReqColidxFor;
								_CPCache[_i].wColBack := IFsvCPCache.In.wReqColidxBack;

								_enSave := cs_SaveCreateCSV;

								_enCmd := cs_CmdSave;

							ELSE

								IFsvCPCache.Out.wCmdResponse := SVCPCACHE_STAT_CATEGORYNOTEXIST;
								_enCmd := cs_CmdWaitForNoCommand;

							END_IF

						ELSE

							IFsvCPCache.Out.wCmdResponse := SVCPCACHE_STAT_INVALIDCATEGORY;
							_enCmd := cs_CmdWaitForNoCommand;

						END_IF

					ELSE

						IFsvCPCache.Out.wCmdResponse := SVCPCACHE_STAT_CATEGORYLISTEMPTY;
						_enCmd := cs_CmdWaitForNoCommand;

					END_IF

				SVCPCACHE_CMD_DELETECATEGORY:

					_wCmd := SVCPCACHE_CMD_DELETECATEGORY;

					IF IFsvCPCache.Out.wCntRelations > 0 THEN

						_TrimCat(sCategory := IFsvCPCache.In.sReqCategory);
						_sCategory := _TrimCat.sOutCategory;

						IF _sCategory <> '' THEN

							_xCategoryExist := FALSE;

							FOR _i := 1 TO SVCPCACHE_CNT_RELATIONS DO

								IF _CPCache[_i].dtTimeStamp = USINT_TO_DT(0) THEN
									EXIT;
								ELSIF _CPCache[_i].sCategory = _sCategory THEN
									_xCategoryExist := TRUE;
									EXIT;
								END_IF

							END_FOR

							IF _xCategoryExist THEN

								IF _i < IFsvCPCache.Out.wCntRelations THEN

									brsmemmove(ADR(_CPCache[_i]), ADR(_CPCache[_i+1]), SIZEOF(_CPCache[1])*(IFsvCPCache.Out.wCntRelations-_i) );

								END_IF

								brsmemset(ADR(_CPCache[IFsvCPCache.Out.wCntRelations]), 0, SIZEOF(_CPCache[1]));

								IFsvCPCache.Out.wCntRelations := IFsvCPCache.Out.wCntRelations - 1;

								_enSave := cs_SaveCreateCSV;

								_enCmd := cs_CmdSave;

							ELSE

								IFsvCPCache.Out.wCmdResponse := SVCPCACHE_STAT_CATEGORYNOTEXIST;
								_enCmd := cs_CmdWaitForNoCommand;

							END_IF

						ELSE

							IFsvCPCache.Out.wCmdResponse := SVCPCACHE_STAT_INVALIDCATEGORY;
							_enCmd := cs_CmdWaitForNoCommand;

						END_IF

					ELSE

						IFsvCPCache.Out.wCmdResponse := SVCPCACHE_STAT_CATEGORYLISTEMPTY;
						_enCmd := cs_CmdWaitForNoCommand;

					END_IF

				SVCPCACHE_CMD_SETOFFSET:

					IFsvCPCache.Out.wListOffset := IFsvCPCache.In.wSetOffset;
					_actFillCPList;

					IFsvCPCache.Out.wCmdResponse := SVCPCACHE_CMD_SETOFFSET;
					_enCmd := cs_CmdWaitForNoCommand;

				SVCPCACHE_CMD_RESTORE:

					IF _enImport = cs_ImpIdle THEN

						_sDevice := IFsvCPCache.In.sImpDevice;
						_sPathFile := CONCAT(IFsvCPCache.In.sImpPath,_SVCPCACHE_CSV_FILE);

						IFsvCPCache.Out.wCmdResponse := KG_STAT_BUSY;
						_wCmd := SVCPCACHE_CMD_RESTORE;

						_enCmd := cs_CmdImport;

						_enImport := cs_ImpStart;

					END_IF

				ELSE

					IFsvCPCache.Out.wCmdResponse := KG_CMDSTAT_NOTVALID;
					_enCmd := cs_CmdWaitForNoCommand;

			END_CASE

		cs_CmdImport:

			(* ACTION*)

			_actCPImport;

			IF _enImport = cs_ImpRdyFault THEN

				// Einlesen mit Fehler abgebrochen
				_xCacheInitReady := FALSE;

				_enImport := cs_ImpIdle;

				IFsvCPCache.Out.wCmdResponse := SVCPCACHE_STAT_FILENOTFOUND;
				_enCmd := cs_CmdWaitForNoCommand;

			ELSIF _enImport = cs_ImpRdySuccess THEN

				// Erfolgreich eingelesen
				_xCacheReady := TRUE;

				IFsvCPCache.Out.xListReady := TRUE;
				IFsvCPCache.Out.wCntRelations := _wCntRelations;

				_enImport := cs_ImpIdle;

				// Liste füllen
				IFsvCPCache.Out.wListOffset := 0;

				_enSave := cs_SaveCreateCSV;
				_enCmd := cs_CmdSave;

			END_IF

		cs_CmdSave:

			IF _enSave = cs_SaveRdySuccess THEN

				_actFillCPList;

				_enSave := cs_SaveIdle;

				IFsvCPCache.Out.wCmdResponse := _wCmd;
				_enCmd := cs_CmdWaitForNoCommand;

			ELSIF _enSave = cs_SaveRdyFault THEN

				_enSave := cs_SaveIdle;

				IFsvCPCache.Out.wCmdResponse := _wSaveCSVstatus;
				_enCmd := cs_CmdWaitForNoCommand;

			END_IF

		cs_CmdWaitForDB:

			IF IFhlDFII.In.ReqProgByCat.wRequest = 0 AND IFhlDFII.Out.RespProgByCat.wResponse = 0 THEN

				IFhlDFII.In.ReqProgByCat.sCategoryNo_In := IFsvCPCache.In.sReqCategory;
				IFhlDFII.In.ReqProgByCat.wRequest		:= 2;

			ELSIF IFhlDFII.In.ReqProgByCat.wRequest = 2 AND IFhlDFII.Out.RespProgByCat.wResponse = 2 THEN

				_DTGetTime(enable := TRUE);

				IFsvCPCache.Out.rRespSoilFactor 		:= IFhlDFII.Out.RespProgByCat.rSoilfactor;
				IFsvCPCache.Out.utfRespCategoryName 	:= STRING_TO_WSTRING(IFhlDFII.Out.RespProgByCat.sCategoryName);
				IFsvCPCache.Out.wRespColidxBack			:= IFhlDFII.Out.RespProgByCat.wColorIdxBack;
				IFsvCPCache.Out.wRespColidxFor			:= IFhlDFII.Out.RespProgByCat.wColorIdxFor;
				IFsvCPCache.Out.wRespLoadrate			:= IFhlDFII.Out.RespProgByCat.wLoadrate;
				IFsvCPCache.Out.wRespProgramNo			:= IFhlDFII.Out.RespProgByCat.bProgramNo;

				FOR _i := 1 TO IFmnParam.Out.Edit.wCntNamelist DO

					IF IFmnParam.Out.Edit.wNameListNo[_i] = IFsvCPCache.Out.wRespProgramNo THEN
						IFsvCPCache.Out.utfRespProgramName := IFmnParam.Out.Edit.utfNameListName[_i];
						EXIT;
					END_IF

				END_FOR

				IFsvCPCache.Out.wRespFromDB				:= SVCPCACHE_DBREQ_DFII;

				IF _xCategoryExist AND
					_CPCache[_wCategoryIdx].utfCategoryName = IFsvCPCache.Out.utfRespCategoryName AND
					_CPCache[_wCategoryIdx].rSoilfactor = IFsvCPCache.Out.rRespSoilFactor AND
					_CPCache[_wCategoryIdx].wLoadrate = IFsvCPCache.Out.wRespLoadrate AND
					_CPCache[_wCategoryIdx].wColBack = IFsvCPCache.Out.wRespColidxBack AND
					_CPCache[_wCategoryIdx].wColFor = IFsvCPCache.Out.wRespColidxFor AND
					_CPCache[_wCategoryIdx].wProgramNo =  IFsvCPCache.Out.wRespProgramNo THEN

					// Lokale Daten sind gleich den Daten aus der Datenbank

					IFsvCPCache.Out.wCmdResponse			:= SVCPCACHE_CMD_GETPROG;
					_enCmd := cs_CmdWaitForNoCommand;

				ELSIF _xCategoryExist THEN

					// Lokale Daten werden aktualisiert

					_CPCache[_wCategoryIdx].utfCategoryName := STRING_TO_WSTRING(IFhlDFII.Out.RespProgByCat.sCategoryName);
					_CPCache[_wCategoryIdx].rSoilfactor 	:= IFhlDFII.Out.RespProgByCat.rSoilfactor;
					_CPCache[_wCategoryIdx].wLoadrate 		:= IFhlDFII.Out.RespProgByCat.wLoadrate;
					_CPCache[_wCategoryIdx].wColBack 		:= IFhlDFII.Out.RespProgByCat.wColorIdxBack;
					_CPCache[_wCategoryIdx].wColFor 		:= IFhlDFII.Out.RespProgByCat.wColorIdxFor;
					_CPCache[_wCategoryIdx].wProgramNo 		:= IFhlDFII.Out.RespProgByCat.bProgramNo;
					_CPCache[_wCategoryIdx].dtTimeStamp		:= _DTGetTime.DT1;

					_wCmd := SVCPCACHE_CMD_GETPROG;
					_enSave := cs_SaveCreateCSV;
					_enCmd := cs_CmdSave;

				ELSE

					// Es wird versucht eine neue Kategorie in den lokalen Speicher abzulegen

					IF IFsvCPCache.Out.wCntRelations < SVCPCACHE_CNT_RELATIONS THEN

						FOR _i := 1 TO SVCPCACHE_CNT_RELATIONS DO

							IF _CPCache[_i].dtTimeStamp = USINT_TO_DT(0) THEN

								_CPCache[_i].dtTimeStamp 		:= _DTGetTime.DT1;
								_CPCache[_i].sCategory 			:= _sCategory;
								_CPCache[_i].utfCategoryName 	:= STRING_TO_WSTRING(IFhlDFII.Out.RespProgByCat.sCategoryName);
								_CPCache[_i].wProgramNo 		:= IFhlDFII.Out.RespProgByCat.bProgramNo;
								_CPCache[_i].rSoilfactor 		:= IFhlDFII.Out.RespProgByCat.rSoilfactor;
								_CPCache[_i].wLoadrate 			:= IFhlDFII.Out.RespProgByCat.wLoadrate;
								_CPCache[_i].wColFor 			:= IFhlDFII.Out.RespProgByCat.wColorIdxFor;
								_CPCache[_i].wColBack 			:= IFhlDFII.Out.RespProgByCat.wColorIdxBack;

								IFsvCPCache.Out.wCntRelations := IFsvCPCache.Out.wCntRelations + 1;

								EXIT;

							ELSIF brsstrcmp(ADR(_CPCache[_i].sCategory),ADR(_sCategory)) > 0 THEN

								brsmemmove(ADR(_CPCache[_i+1]), ADR(_CPCache[_i]), SIZEOF(_CPCache[1])*(IFsvCPCache.Out.wCntRelations-_i+1) );

								_CPCache[_i].dtTimeStamp 		:= _DTGetTime.DT1;
								_CPCache[_i].sCategory 			:= _sCategory;
								_CPCache[_i].utfCategoryName 	:= STRING_TO_WSTRING(IFhlDFII.Out.RespProgByCat.sCategoryName);
								_CPCache[_i].wProgramNo 		:= IFhlDFII.Out.RespProgByCat.bProgramNo;
								_CPCache[_i].rSoilfactor 		:= IFhlDFII.Out.RespProgByCat.rSoilfactor;
								_CPCache[_i].wLoadrate 			:= IFhlDFII.Out.RespProgByCat.wLoadrate;
								_CPCache[_i].wColFor 			:= IFhlDFII.Out.RespProgByCat.wColorIdxFor;
								_CPCache[_i].wColBack 			:= IFhlDFII.Out.RespProgByCat.wColorIdxBack;

								IFsvCPCache.Out.wCntRelations := IFsvCPCache.Out.wCntRelations + 1;

								EXIT;

							END_IF

						END_FOR

						_wCmd := SVCPCACHE_CMD_GETPROG;
						_enSave := cs_SaveCreateCSV;
						_enCmd := cs_CmdSave;

					ELSE

						// Kein Platz für eine neue Kategorie

						IFsvCPCache.Out.wCmdResponse			:= SVCPCACHE_CMD_GETPROG;
						_enCmd := cs_CmdWaitForNoCommand;

					END_IF

				END_IF

				IFhlDFII.In.ReqProgByCat.wRequest		:= 0;

			ELSIF IFhlDFII.In.ReqProgByCat.wRequest = 2 AND IFhlDFII.Out.RespProgByCat.wResponse <> 65535 AND IFhlDFII.Out.RespProgByCat.wResponse <> 0 THEN

				IF _xCategoryExist THEN

					IFsvCPCache.Out.rRespSoilFactor 		:= _CPCache[_wCategoryIdx].rSoilfactor;
					IFsvCPCache.Out.utfRespCategoryName		:= _CPCache[_wCategoryIdx].utfCategoryName;
					IFsvCPCache.Out.wRespColidxBack			:= _CPCache[_wCategoryIdx].wColBack;
					IFsvCPCache.Out.wRespColidxFor			:= _CPCache[_wCategoryIdx].wColFor;
					IFsvCPCache.Out.wRespLoadrate			:= _CPCache[_wCategoryIdx].wLoadrate;
					IFsvCPCache.Out.wRespProgramNo			:= _CPCache[_wCategoryIdx].wProgramNo;

					FOR _i := 1 TO IFmnParam.Out.Edit.wCntNamelist DO

						IF IFmnParam.Out.Edit.wNameListNo[_i] = IFsvCPCache.Out.wRespProgramNo THEN
							IFsvCPCache.Out.utfRespProgramName := IFmnParam.Out.Edit.utfNameListName[_i];
							EXIT;
						END_IF

					END_FOR

					IFsvCPCache.Out.wCmdResponse 			:= SVCPCACHE_CMD_GETPROG;

				ELSE

					IFsvCPCache.Out.wCmdResponse			:= IFhlDFII.Out.RespProgByCat.wResponse;

				END_IF

				IFhlDFII.In.ReqProgByCat.wRequest		:= 0;
				_enCmd := cs_CmdWaitForNoCommand;

			END_IF

		cs_CmdWaitForNoCommand:

			IF IFsvCPCache.In.wCmd = KG_CMD_NOCOMMAND THEN

				IFsvCPCache.Out.wCmdResponse := KG_STAT_OK;

				_enCmd := cs_CmdIdle;

			END_IF

	END_CASE

END_ACTION
```

#### _actFillCPList.st
```iecst
(********************************************************************
 * COPYRIGHT -- Herbert Kannegiesser GmbH
 ********************************************************************
 * Program: svCPCache
 * File: _actFillCPList.st
 * Author: hunholz
 * Created: March 30, 2012
 ********************************************************************
 * Implementation of program svCPCache
 ********************************************************************)

(* Add a new action to your IEC program or library *)
ACTION _actFillCPList:

	IF _xCacheReady AND SVCPCACHE_CNT_LISTRELATIONS > 0 THEN

		IF SVCPCACHE_CNT_RELATIONS > SVCPCACHE_CNT_LISTRELATIONS THEN

			IFsvCPCache.Out.wListOffset := MIN(IFsvCPCache.Out.wListOffset, SVCPCACHE_CNT_RELATIONS-SVCPCACHE_CNT_LISTRELATIONS);

		ELSE

			IFsvCPCache.Out.wListOffset := 0;

		END_IF

		IFsvCPCache.Out.wListCnt := 0;
		brsmemset(ADR(IFsvCPCache.Out.sListCategory), 0, SIZEOF(IFsvCPCache.Out.sListCategory));
		brsmemset(ADR(IFsvCPCache.Out.utfListCategoryname), 0, SIZEOF(IFsvCPCache.Out.utfListCategoryname));
		brsmemset(ADR(IFsvCPCache.Out.utfListProgramName), 0, SIZEOF(IFsvCPCache.Out.utfListProgramName));
		brsmemset(ADR(IFsvCPCache.Out.wListProgramNo), 0, SIZEOF(IFsvCPCache.Out.wListProgramNo));

		FOR _wfcli := 1 TO SVCPCACHE_CNT_LISTRELATIONS DO

			IF _wfcli + IFsvCPCache.Out.wListOffset <= SVCPCACHE_CNT_RELATIONS THEN

				IF _CPCache[_wfcli + IFsvCPCache.Out.wListOffset].dtTimeStamp > USINT_TO_DT(0) THEN

					IFsvCPCache.Out.sListCategory[_wfcli] := _CPCache[_wfcli + IFsvCPCache.Out.wListOffset].sCategory;
					IFsvCPCache.Out.wListProgramNo[_wfcli] := _CPCache[_wfcli + IFsvCPCache.Out.wListOffset].wProgramNo;
					IFsvCPCache.Out.utfListCategoryname[_wfcli] := _CPCache[_wfcli + IFsvCPCache.Out.wListOffset].utfCategoryName;

					FOR _wfclj := 1 TO IFmnParam.Out.Edit.wCntNamelist DO

						IF IFmnParam.Out.Edit.wNameListNo[_wfclj] = IFsvCPCache.Out.wListProgramNo[_wfcli] THEN
							IFsvCPCache.Out.utfListProgramName[_wfcli] := IFmnParam.Out.Edit.utfNameListName[_wfclj];
							EXIT;
						END_IF

					END_FOR

					IFsvCPCache.Out.wListCnt := IFsvCPCache.Out.wListCnt + 1;

				ELSE

					EXIT;

				END_IF

			END_IF

		END_FOR

	END_IF

END_ACTION
```

#### _actSaveCSV.st
```iecst
(********************************************************************
 * COPYRIGHT -- Herbert Kannegiesser GmbH
 ********************************************************************
 * Program: svCPCache
 * File: _actSaveCSV.st
 * Author: hunholz
 * Created: March 30, 2012
 ********************************************************************
 * Implementation of program svCPCache
 ********************************************************************)

(* Schrittkette zum Speichern der Kategorie-Programm-Zuordnung *)
ACTION _actSaveCSV:

	_wSaveCSVstatus := ERR_OK;

	CASE _enSave OF

		cs_SaveIdle:

			// Tue nichts

		cs_SaveCreateCSV:

			_SaveMemPartAlloc(enable := TRUE, ident := _MemPartCreate.ident , len := _lMemLen);
			_lWriteSize := 0;

			IF _SaveMemPartAlloc.status = ERR_OK THEN

				_WriteBOM(enable := TRUE, pMem := _SaveMemPartAlloc.mem, lMaxSize := _lMemLen, lSize := _lWriteSize);

				// Kopfdaten schreiben
				_WriteComment(enable := TRUE, pMem := _SaveMemPartAlloc.mem, lMaxSize := _lMemLen, sComment := CONCAT('svCPCache Version: ',svCPCacheStatAd.sPkgVersion) , lSize := _lWriteSize);
				_WriteNewLine(enable := TRUE, pMem := _SaveMemPartAlloc.mem, lMaxSize := _lMemLen, lSize := _lWriteSize);

				_MachineNoRow.utfMachineNo := IFmnParam.Out.utfMachineNumber;
				_WriteMachineNo(enable := TRUE, pMem := _SaveMemPartAlloc.mem, lMaxSize := _lMemLen, MachineNoRow := _MachineNoRow, lSize := _lWriteSize);

				_WriteNewLine(enable := TRUE, pMem := _SaveMemPartAlloc.mem, lMaxSize := _lMemLen, lSize := _lWriteSize);

				_DTGetTime(enable := TRUE);
				_HeaderTimeRow.dtTimestamp := _DTGetTime.DT1;

				_WriteTimeStamp(enable := TRUE, pMem := _SaveMemPartAlloc.mem, lMaxSize := _lMemLen, TimeRow := _HeaderTimeRow, lSize := _lWriteSize);

				_WriteNewLine(enable := TRUE, pMem := _SaveMemPartAlloc.mem, lMaxSize := _lMemLen, lSize := _lWriteSize);

				FOR _sci := 1 TO SVCPCACHE_CNT_RELATIONS DO

					IF _CPCache[_sci].dtTimeStamp <> USINT_TO_DT(0) AND _CPCache[_sci].sCategory <> '' THEN

						_WriteCP(enable := TRUE, pMem := _SaveMemPartAlloc.mem, lMaxSize := _lMemLen, CPRow := _CPCache[_sci], lSize := _lWriteSize);

					END_IF

				END_FOR

				_sPathFile := CONCAT(_SVCPCACHE_CSV_PATH,_SVCPCACHE_CSV_FILE);

				_enSave := cs_SaveDeleteFile;

			ELSE

				_wSaveCSVstatus := SVCPCACHE_STAT_MEMALLOC;
				_enSave := cs_SaveRdyFault;

			END_IF

		cs_SaveDeleteFile:

			_FileDelete(enable := TRUE, pDevice := ADR(KG_DEVICE_COMPACTFLASH), pName := ADR(_sPathFile));

			IF _FileDelete.status <> ERR_FUB_BUSY THEN

				_enSave := cs_SaveCreateFile;

			END_IF

		//==============================================
		// Exportdatei erzeugen
		//==============================================
		cs_SaveCreateFile:

			_FileCreate(enable := TRUE, pDevice := ADR(KG_DEVICE_COMPACTFLASH), pFile := ADR(_sPathFile) );

			IF _FileCreate.status = ERR_OK THEN

				_enSave := cs_SaveWriteFile;

			ELSIF _FileCreate.status <> ERR_FUB_BUSY THEN

				_SaveMemPartFree(enable := TRUE, ident := _MemPartCreate.ident, mem := _SaveMemPartAlloc.mem);

				_wSaveCSVstatus := SVCPCACHE_STAT_CREATEFILE;
				_enSave := cs_SaveRdyFault;

			END_IF

		//==============================================
		// Exportdatei öffnen
		//==============================================
		cs_SaveOpenFile:

			_FileOpen(enable := TRUE, pDevice := ADR(KG_DEVICE_COMPACTFLASH), pFile := ADR(_sPathFile), mode := fiWRITE_ONLY);

			IF _FileOpen.status = ERR_OK THEN

				_enSave := cs_SaveWriteFile;

			ELSIF _FileOpen.status <> ERR_FUB_BUSY THEN

				_SaveMemPartFree(enable := TRUE, ident := _MemPartCreate.ident, mem := _SaveMemPartAlloc.mem);

				_wSaveCSVstatus := SVCPCACHE_STAT_OPENFILE;
				_enSave := cs_SaveRdyFault;

			END_IF

		//==============================================
		// Exportdatei schreiben
		//==============================================
		cs_SaveWriteFile:

			_FileWrite(enable := TRUE, ident := _FileCreate.ident, offset := 0, pSrc :=_SaveMemPartAlloc.mem, len := _lWriteSize);

			IF _FileWrite.status = ERR_OK THEN

				_SaveMemPartFree(enable := TRUE, ident := _MemPartCreate.ident, mem := _SaveMemPartAlloc.mem);
				_enSave := cs_SaveCloseFile;

			ELSIF _FileWrite.status <> ERR_FUB_BUSY THEN

				_SaveMemPartFree(enable := TRUE, ident := _MemPartCreate.ident, mem := _SaveMemPartAlloc.mem);

				_wSaveCSVstatus := SVCPCACHE_STAT_WRITEFILE;
				_enSave := cs_SaveCloseFile;

			END_IF

		//==============================================
		// Exportdatei schließen
		//==============================================
		cs_SaveCloseFile:

			_FileClose(enable := TRUE, ident := _FileCreate.ident);

			IF _FileClose.status <> ERR_FUB_BUSY THEN

				IF _wSaveCSVstatus = ERR_OK THEN

					_enSave := cs_SaveRdySuccess;

				ELSE

					_enSave := cs_SaveRdyFault;

				END_IF

			END_IF

		cs_SaveRdyFault:

			// Mit Fehler beendet

		cs_SaveRdySuccess:

			// Erfolgreich beendet

	END_CASE

END_ACTION
```

#### _TrimCategory.st - Entfernt führende Nullen und Leerzeichen, sowie folgende Leerzeichen
```iecst
(********************************************************************
 * COPYRIGHT -- Herbert Kannegiesser GmbH
 ********************************************************************
 * Program: svCPCache
 * File: _TrimCategory.st
 * Author: hunholz
 * Created: March 30, 2012
 ********************************************************************
 * Implementation of program svCPCache
 ********************************************************************)

(* Entfernt führende Nullen und Leerzeichen, sowie folgende Leerzeichen *)
FUNCTION_BLOCK _TrimCategory

	sOutCategory := sCategory;

	IF LEN(sOutCategory) > 0 THEN
		REPEAT
			_iFound := FIND(sOutCategory,' ');

			IF _iFound <> 0 THEN
				sOutCategory := DELETE(sOutCategory,1,_iFound);
			END_IF

			UNTIL
			_iFound = 0 OR LEN(sOutCategory) = 0
		END_REPEAT
	END_IF

	//Bug 689: Eine Null muss stehen bleiben
	IF LEN(sOutCategory) > 1 THEN
		REPEAT
			_iFound := FIND(sOutCategory,'0');

			IF _iFound = 1 THEN
				sOutCategory := DELETE(sOutCategory,1,_iFound);
			END_IF

			UNTIL
			_iFound <> 1 OR LEN(sOutCategory) = 1
		END_REPEAT
	END_IF

END_FUNCTION_BLOCK
```

#### svCPCache.fun
```iecst
(********************************************************************
 * COPYRIGHT -- Herbert Kannegiesser GmbH
 ********************************************************************
 * Program: svCPCache
 * File: svCPCache.fun
 * Author: hunholz
 * Created: March 30, 2012
 ********************************************************************
 * Functions and function blocks of program svCPCache
 ********************************************************************)

FUNCTION_BLOCK _TrimCategory (*Entfernt führende Nullen und Leerzeichen, sowie folgende Leerzeichen*)
	VAR_INPUT
		sCategory : STRING[11];
	END_VAR
	VAR_OUTPUT
		sOutCategory : STRING[11];
	END_VAR
	VAR
		_iFound : INT;
	END_VAR
END_FUNCTION_BLOCK
```

### svCPCacheHistory.txt
```
0.02.0	Start der Historie
0.03.0	19.06.2012	Kategorie 0 lässt sich nicht anlegen. Bug 689 behoben.
0.03.1	26.06.2012	Warnung unterdrückt
0.03.2	17.07.2012	Bugfix - Filehandles wurden nach einem Create nicht freigegeben.
```

### hlKanLink.typ - Global data types
```iecst
(********************************************************************
 * COPYRIGHT -- Bernecker + Rainer
 ********************************************************************
 * File: Global.typ
 * Author: Bernecker + Rainer
 * Created: June 02, 2008
 ********************************************************************
 * Global data types of project LibAsUDP
 ********************************************************************)

TYPE
	hlKanLinkStatAd_typ : 	STRUCT
		sPkgVersion : STRING[11];
	END_STRUCT;
END_TYPE
```

### hlKanLink.var - Global variables
```iecst
(********************************************************************
 * COPYRIGHT -- Bernecker + Rainer
 ********************************************************************
 * File: Global.var
 * Author: Bernecker + Rainer
 * Created: June 02, 2008
 ********************************************************************
 * Global variables of project LibAsUDP
 ********************************************************************)
VAR
	hlKanLinkStatAd : hlKanLinkStatAd_typ;
	IFhlKanLink : IFhlKanLink_Typ;
END_VAR
(*Konstanten*)
VAR CONSTANT
	HLKANLINK_MSG_NO_STRUCDEF : UINT := 60000;
END_VAR
VAR
	IFhlKL_Visu : IFhlKLVisu_typ;
END_VAR
```

### Program Logical/Standard/Kanlink/KGFramework/Pkg_hlKanLink/hlKanLink (IEC) - Kanlink Task

#### KanLink.typ - Local data types
```iecst
(********************************************************************
 * COPYRIGHT -- Herbert Kannegiesser GmbH
 ********************************************************************
 * Program: WetLink
 * File: WetLink.typ
 * Author: stahlhut
 * Created: December 23, 2011
 ********************************************************************
 * Local data types of program WetLink
 ********************************************************************)

TYPE
	ErrLog_typ : 	STRUCT
		wErrorNo : UINT;
		lAttr1 : UDINT;
		lAttr2 : UDINT;
	END_STRUCT;
END_TYPE
```

#### KanLink.var - Local variables
```iecst
(********************************************************************
 * COPYRIGHT -- Herbert Kannegiesser GmbH
 ********************************************************************
 * Program: WetLink
 * File: WetLink.var
 * Author: stahlhut
 * Created: December 23, 2011
 ********************************************************************
 * Local variables of program WetLink
 ********************************************************************)
VAR
	_AsArLogCreate : AsArLogCreate;
	_AsArLogGetInfo : AsArLogGetInfo;
	_dClient : REFERENCE TO KL_ClientListe_typ;
	_dCltIf : REFERENCE TO IF_Client_typ;
	_dSrvIf : REFERENCE TO IF_Server_typ;
END_VAR
VAR CONSTANT
	_HLKANLINK_IDX_STRUCDEF_RESP_0 : UINT := 1;
	_HLKANLINK_MAX_IDX_DEFSTRUC : UINT := 5;
END_VAR
VAR
	_i : UINT;
	_iCltIdx : INT;
	_iCltRespCnt : INT;
	_ifDummy : IF_Client_typ;
	_iIdxFound : INT;
END_VAR
VAR RETAIN
	_iLastCltIdx : UINT;
	_iLastMuCltIdx : UINT;
END_VAR
VAR
	_iLastServerIdx : UINT;
	_iMuCltIdx : INT;
	_InsertRB : kgRBinsert;
	_k : UINT;
	_kgArLogWrite : kgArLogWrite;
	_kgRBcreateKanLinklog : kgRBcreate;
	_lAdr : UDINT;
	_lLen : UDINT;
	_lMemIdent : UDINT;
	_LogEntry : ErrLog_typ;
	_LogEntryIn : ErrLog_typ;
	_lPtrStrucDef : ARRAY[0..5] OF UDINT;
	_lPtrStrucLen : ARRAY[0..5] OF UDINT;
	_lTempMemIdent : UDINT;
	_MemAlloc : AsMemPartAllocClear;
	_MemAllocTemp : AsMemPartAllocClear;
	_MemFreeTemp : AsMemPartFree;
	_MemPartCreate : AsMemPartCreate;
	_ptrIndex : REFERENCE TO KL_ServerListe_typ;
	_ReadRB : kgRBread;
	_sClientIPAdr : STRING[16];
	_sDebString : REFERENCE TO STRING[31];
	_sName : STRING[80];
	_sPkgName : STRING[11];
	_state : USINT;
	_tcnr : SINT;
	_VerStruc : MoVerStruc_typ;
	_wClt : UINT;
	_wDebIdx : UINT;
	_wDebOffset : UINT;
	_wLogStep : UINT;
	_wPtrRBloc : UINT;
	_wPtrRBread : UINT;
	_wPtrRBstart : UINT;
	_wPtrRBwrite : UINT;
	_wSrv : UINT;
	_wStatus : UINT;
	_xAdrErr : BOOL;
	_xAdrOK : BOOL;
	_xCheckClt : BOOL;
	_xCltFound : BOOL;
	_xIdxFound : BOOL;
	_xInitOK : BOOL;
	_xRBReady : BOOL;
	_xSaveConfig : BOOL;
	_xSendNow : BOOL;
	_xServerFound : BOOL;
	Kanlink : KanLink_FB;
	KL_SaveConfDO_0 : KL_SaveConfDO;
	WL_ErrorNr : UINT;
END_VAR
```

#### KanLinkCyclic.st - Cyclic code
```iecst
(********************************************************************
 * COPYRIGHT -- Herbert Kannegiesser GmbH
 ********************************************************************
 * Program: KanLink
 * File: KanLinkCyclic.st
 * Author: stahlhut
 * Created: December 23, 2011
 ********************************************************************
 * Implementation of program WetLink
 ********************************************************************)

(*

	Falls ohne Framework gearbeitet werden soll in den Eigenschaften der Task hlKanLink (Config. View Cpu.sw)
	im Tab. Compiler im Feld "Additional build options:" -D HLKANLINK_AUTONOM  eintragen
	Dazu das Package KanLinkAutonom importieren

*)

PROGRAM _CYCLIC

// Struktur für Visualisierung füllen

IFhlKL_Visu.out.iCycleTime := Kanlink._iCycleTime;
IFhlKL_Visu.out.step := Kanlink.Step;
IFhlKL_Visu.out.udNetId := Kanlink.udNetID;
IFhlKL_Visu.out.udpOpenStatus := Kanlink.udp.open.status;
IFhlKL_Visu.out.udpRecStatus := Kanlink.udp.rec.status;
IFhlKL_Visu.out.udpSendStatus := Kanlink.udp.send.status;
_wClt := LIMIT(0,IFhlKL_Visu.in.iCltNr,HLKANLINK_MAX_CLIENTCONNS);
_wSrv := LIMIT(0,IFhlKL_Visu.in.iServerNr,HLKANLINK_MAX_SERVERCONNS);
IFhlKL_Visu.out.client := Kanlink.ClientListe[_wClt];
IFhlKL_Visu.out.server := Kanlink.ServerListe[_wSrv];

// Commando von der Visu verarbeiten
// Commando nur setzen wenn CmdResp = 0
// aufrufer muss nach ausführung cmdNr wieder auf 0 setzen!
IF IFhlKL_Visu.in.cmdNr <> IFhlKL_Visu.out.cmdResp THEN
	CASE IFhlKL_Visu.in.cmdNr OF
		0: IFhlKL_Visu.out.cmdResp := 0;
		1: // Neustart
			IFhlKL_Visu.out.cmdResp := 1;
			Kanlink.Step := 1;
		2: // Neustart mit lastId = 1
			Kanlink._uiLastId := 1;
			IFhlKL_Visu.out.cmdResp := 1;
			Kanlink.Step := 2;
		ELSE
			// unbekanntes Commando
			IFhlKL_Visu.out.cmdResp := 16#7FFF;

	END_CASE;
END_IF;

#ifndef HLKANLINK_AUTONOM // Logging nur mit kg-Framework

	// ===========================
	// Logging
	// ===========================

	IF _xRBReady THEN

		CASE _wLogStep OF

			0:
				_ReadRB(wPtrRead := _wPtrRBread, wPtrStart := _wPtrRBstart, wPtrWrite := _wPtrRBwrite);

				IF _ReadRB.wStatus = ERR_OK THEN

					CASE _LogEntry.wErrorNo OF

						0:
							_kgArLogWrite.text := 'OK';

						HLKANLINK_MSG_NO_STRUCDEF:

							_kgArLogWrite.text := 'Create Strucdefinition failed : {##AttrVar1} / {##AttrVar2}';
							_kgArLogWrite.var1 := _LogEntry.lAttr1;

						ELSE

							_kgArLogWrite.text := UINT_TO_STRING(_LogEntry.wErrorNo);
							_kgArLogWrite.text := CONCAT(_kgArLogWrite.text, ' : {##AttrVar1} / {##AttrVar2}');
							_kgArLogWrite.var1 := _LogEntry.lAttr1;
							_kgArLogWrite.var2 := _LogEntry.lAttr2;

					END_CASE

					_wLogStep := 1;

				END_IF

			1:
				_kgArLogWrite();

				IF _kgArLogWrite.status <> ERR_FUB_BUSY THEN

					_wLogStep := 0;

				END_IF

		END_CASE

	END_IF

	IF _wDebIdx >= 0 AND _wDebIdx <= _HLKANLINK_MAX_IDX_DEFSTRUC THEN

		IF _lPtrStrucDef[_wDebIdx] > 0 THEN

			_sDebString ACCESS _lPtrStrucDef[_wDebIdx] + _wDebOffset;

		END_IF

	END_IF

#endif

	// =======================================================================

	IF _xInitOK THEN

		IF _xSaveConfig THEN
			KL_SaveConfDO_0(adrName :=ADR('KL_Conf') , adrDaten := ADR(IFhlKanLink.Parameter), len := SIZEOF( IFhlKanLink.Parameter));
			IF KL_SaveConfDO_0.status <> ERR_FUB_BUSY THEN // fertig
				_xSaveConfig := FALSE;
			END_IF;
		END_IF;

		IF EDGEPOS(IFhlKanLink.in.xRun ) THEN
			IF Kanlink.Step = 0 THEN
				Kanlink.Step := 1;
			END_IF;
		END_IF;
		IF EDGENEG(IFhlKanLink.in.xRun) THEN // stoppen
			IF Kanlink.Step <> 0 THEN
				Kanlink.Step := 20;
			END_IF;
		END_IF;

		IF IFhlKanLink.in.xRestart THEN
			Kanlink.Step := 1;
			IFhlKanLink.in.xRestart := 0;
		END_IF;

		IFhlKanLink.xError := (Kanlink.Step = 200);

		CASE Kanlink.Step OF

			0: //nix tun

			100: // Error nr in Logger eintragen

				Kanlink.Step := 200;

			200: // Auf User warten

			1: // init

				Kanlink.KLLib_Init_0(enable := 1, adrServer := ADR(Kanlink),adrInterface := ADR(IFhlKanLink));
				IF Kanlink.KLLib_Init_0.status = ERR_OK THEN
					Kanlink.Step := 10;
				ELSIF Kanlink.KLLib_Init_0.status <> ERR_FUB_BUSY THEN // fehler
					WL_ErrorNr := 10;
					Kanlink.Step := 100;

					IF _xRBReady THEN

						_LogEntryIn.wErrorNo := 10;
						_InsertRB(wPtrStart := _wPtrRBstart, wPtrRead := _wPtrRBread, wPtrWrite := _wPtrRBwrite);

					END_IF

				END_IF;

			10: // Kanlink Run

			20: // Kanlink schliessen

				Kanlink.udp.close.enable := 1;
				Kanlink.udp.close.ident := Kanlink._uiLastId;
				Kanlink.udp.close;
				IF Kanlink.udp.close.status = 0 THEN
					Kanlink.Step := 0;
				ELSIF Kanlink.udp.close.status = ERR_FUB_BUSY THEN

				ELSE
					Kanlink.Step := 100;
				END_IF;

		END_CASE;

		// interne Zustände auf out Struktur legen
		IFhlKanLink.out.iStep  := Kanlink.Step;
		// noch auzufüllen ....
//		IFhlKanLink.out.iError := ??;
//		IFhlKanLink.out.iClientError[0] := ??;
//		IFhlKanLink.out.iServerError[0] := ??;

		// hier beenden wenn zyklus nicht erlaubt
		IF  Kanlink.Step <> 10 THEN
			RETURN;
		END_IF;

		Kanlink;

		// falls Kanlink nix zu tun hat, hier beenden
		IF Kanlink.xReturn THEN
			RETURN;
		END_IF;

		// ------------------------------------------------------------------
		// Falls ein Request eines Clients aufgelaufen ist

		IF Kanlink._xGetServerReq THEN  // Req eines Clients angenommen, bearbeiten

			actGetServerReq;

			Kanlink._xGetServerReq := FALSE;
			Kanlink.udp.rec.enable := 1;

			RETURN;  // Daten sind versendet. Also Ende.

		END_IF;

		// ------------------------------------------------------------------------------
		// falls Response von einem Request kommt:

		IF Kanlink._xGetClientResp THEN // Response auf ClientReq angekommen
			actResponse;

		END_IF;

		// ------------------------------------------------------------------------------
		// Überprüfen ob per Hand bearbeitete Requests versendet werden müssen..

		IF  Kanlink.udp.send.enable = 0 THEN
			_xServerFound := 0;

			FOR _i:=0 TO HLKANLINK_MAX_SERVERCONNS  DO
				_ptrIndex ACCESS ADR(Kanlink.ServerListe[_iLastServerIdx]);
				_dSrvIf ACCESS _ptrIndex.adrInterface;
				IF (_ptrIndex.xReqManually AND (_dSrvIf.iState = 2)) THEN
					_xServerFound := 1;

					_iLastServerIdx := _iLastServerIdx + 1; // testen
					IF _iLastCltIdx > HLKANLINK_MAX_SERVERCONNS THEN
						_iLastServerIdx := 0;
					END_IF;
					EXIT;
					END_IF;
					_iLastServerIdx := _iLastServerIdx + 1; // testen
					IF _iLastServerIdx > HLKANLINK_MAX_SERVERCONNS THEN
					_iLastServerIdx := 0;
				END_IF;

			END_FOR;

			IF _xServerFound THEN
				Kanlink.ServerData.HeaderV1Send[0].Command := _ptrIndex.Cmd + 1;
				Kanlink.ServerData.HeaderV1Send[0].dataFormat := 5;
				Kanlink.ServerData.HeaderV1Send[0].Length := UDINT_TO_UINT( _ptrIndex.RespLength);
				Kanlink.ServerData.HeaderV1Send[0].ReqID := _ptrIndex.iReqID;
				Kanlink.ServerData.HeaderV1Send[0].CmdNr := _ptrIndex.CmdOpt AND 16#00FF;
				_ptrIndex.iConnectionTimer := 0;
				KLLib_SendData(ADR(Kanlink),_ptrIndex.AdrDataResp,_ptrIndex.RespLength,ADR(_ptrIndex.sClientIPAdr),-1,-1,0);
				_dSrvIf.iState := 0;
				RETURN;
			END_IF;
		END_IF;

		IF Kanlink._xSendClient THEN  // hier den Clienten bearbeiten
			_xCltFound := FALSE;
			_iCltIdx := -1;
			_iMuCltIdx := -1;

			FOR _i:=0 TO HLKANLINK_MAX_CLIENTCONNS  DO
				IF (Kanlink.ClientListe[_iLastCltIdx].MuClient >= 0) THEN
					IF ((Kanlink.MuClientListe[Kanlink.ClientListe[_iLastCltIdx].MuClient].bUse = 0) OR (Kanlink.MuClientListe[Kanlink.ClientListe[_iLastCltIdx].MuClient].bUse = 255)) THEN
						_xCheckClt := TRUE;
					ELSE
						_xCheckClt := FALSE;
					END_IF
				ELSE
					_xCheckClt := TRUE;
				END_IF

				IF (_xCheckClt = TRUE) THEN
					_dClient ACCESS ADR(Kanlink.ClientListe[_iLastCltIdx]);
					IF _dClient.adrInterface <> 0 THEN
						_dCltIf ACCESS _dClient.adrInterface;
					ELSE
						_dCltIf ACCESS ADR(_ifDummy);
					END_IF;
						// gefunden wenn kein ReqPend, Commando <> 0 todo gültige Adresse etc...
					IF _dClient.iCycleTime = 0 THEN
						_xSendNow := (_dCltIf.iState = 1) OR (_dCltIf.iState = 4) ; // falls angetickt oder timeout
					ELSE
						_xSendNow := (_dClient.iCycleWait > _dClient.iCycleTime);
					END_IF;
					IF 	(NOT _dClient.xReqPending) AND (_dClient.Cmd <> 0) AND _dClient.xActiv AND (_xSendNow) THEN
			  			_xCltFound := TRUE;
						_iCltIdx := _iLastCltIdx;
						_iLastCltIdx := _iLastCltIdx + 1; // testen
						IF _iLastCltIdx > HLKANLINK_MAX_CLIENTCONNS THEN
				  			_iLastCltIdx := 0;
						END_IF;
						EXIT;
					END_IF;
				END_IF

				_iLastCltIdx := _iLastCltIdx + 1; // testen
				IF _iLastCltIdx > HLKANLINK_MAX_CLIENTCONNS THEN
		  			_iLastCltIdx := 0;
				END_IF;

			END_FOR;

			IF (NOT _xCltFound) THEN
				FOR _i:=0 TO HLKANLINK_MAX_MU_CLIENTCONNS DO
					IF ((Kanlink.MuClientListe[_iLastMuCltIdx].bUse = 1) OR (Kanlink.MuClientListe[_iLastMuCltIdx].bUse = 2)) THEN

						IF Kanlink.ClientListe[Kanlink.MuClientListe[_iLastMuCltIdx].Clients[0]].adrInterface <> 0 THEN
							_dCltIf ACCESS Kanlink.ClientListe[Kanlink.MuClientListe[_iLastMuCltIdx].Clients[0]].adrInterface;
						ELSE
							_dCltIf ACCESS ADR(_ifDummy);
						END_IF;
							// gefunden wenn kein ReqPend, Commando <> 0 todo gültige Adresse etc...
						IF Kanlink.MuClientListe[_iLastMuCltIdx].iCycleTime = 0 THEN
							_xSendNow := (_dCltIf.iState = 1) OR (_dCltIf.iState = 4) ; // falls angetickt oder timeout
						ELSE
							_xSendNow := (Kanlink.MuClientListe[_iLastMuCltIdx].iCycleWait > Kanlink.MuClientListe[_iLastMuCltIdx].iCycleTime);
						END_IF;

						IF 	(NOT Kanlink.MuClientListe[_iLastMuCltIdx].xReqPending) AND Kanlink.MuClientListe[_iLastMuCltIdx].xActiv AND (_xSendNow) THEN
				  			_xCltFound := TRUE;
							_iMuCltIdx := _iLastMuCltIdx;
							_iLastMuCltIdx := _iLastMuCltIdx + 1; // testen
							IF _iLastMuCltIdx > HLKANLINK_MAX_MU_CLIENTCONNS THEN
					  			_iLastMuCltIdx := 0;
							END_IF;
							EXIT;
						END_IF;

					END_IF

					_iLastMuCltIdx := _iLastMuCltIdx + 1; // testen
					IF _iLastMuCltIdx > HLKANLINK_MAX_MU_CLIENTCONNS THEN
			  			_iLastMuCltIdx := 0;
					END_IF;

				END_FOR;
			END_IF

			IF NOT _xCltFound THEN
				Kanlink._xSendClient := FALSE;
				RETURN;

			ELSE

				IF (_iCltIdx >= 0) THEN
					// Client gefunden
					_dClient.iCnt := _dClient.iCnt + 1 ;
					_dClient.iReqId := _dClient.iReqId +1;
					_dClient.TimeOutLeft := _dClient.TimeOut;

					IF _dCltIf.iState = 1 THEN // falls über state dann "schnellwiederholung" aktivieren
						_dClient.iTimeOutCnt := 0; // scharf machen für den nächsten versuch
					END_IF;
					_dCltIf.iState := 2;

					Kanlink.ServerData.HeaderV1Send[0].Command := _dClient.Cmd;
					Kanlink.ServerData.HeaderV1Send[0].CmdNr := _dClient.CmdOpt AND 16#00FF;

					Kanlink.ServerData.HeaderV1Send[0].dataFormat := 5;
					Kanlink.ServerData.HeaderV1Send[0].Length := UDINT_TO_UINT( _dClient.ReqLength);
					Kanlink.ServerData.HeaderV1Send[0].ReqID := _dClient.iReqId;
					Kanlink.ServerData.HeaderV1Send[0].Tag		:= _dCltIf.tag;

// warum ?			KLLib_SendData(ADR(Kanlink),0,                  0,                 ADR(_dClient.sClientAdr),_iCltIdx,-1,KLLIB_REQ);
					KLLib_SendData(ADR(Kanlink),_dClient.AdrDataReq,_dClient.ReqLength,ADR(_dClient.sClientAdr),-1,      -1,KLLIB_REQ);

					_dClient.xReqPending := TRUE;
					_dClient.iCycleWait := 0;

					Kanlink._xSendClient := FALSE;

					RETURN;

				ELSIF (_iMuCltIdx >= 0) THEN

					// Client gefunden
					Kanlink.MuClientListe[_iMuCltIdx].iCnt := Kanlink.MuClientListe[_iMuCltIdx].iCnt + 1;
					Kanlink.MuClientListe[_iMuCltIdx].iReqId := Kanlink.MuClientListe[_iMuCltIdx].iReqId + 1;
					Kanlink.MuClientListe[_iMuCltIdx].TimeOutLeft := Kanlink.MuClientListe[_iMuCltIdx].TimeOut;

					IF _dCltIf.iState = 1 THEN // falls über state dann "schnellwiederholung" aktivieren
						Kanlink.MuClientListe[_iMuCltIdx].iTimeOutCnt := 0; // scharf machen für den nächsten versuch
					END_IF;
					_dCltIf.iState := 2;

					FOR _i := 0 TO KLLIB_MAX_MUL DO

						IF (Kanlink.MuClientListe[_iMuCltIdx].Clients[_i] >= 0) THEN

							Kanlink.ClientListe[Kanlink.MuClientListe[_iMuCltIdx].Clients[_i]].iCnt := Kanlink.MuClientListe[_iMuCltIdx].iCnt;
							Kanlink.ClientListe[Kanlink.MuClientListe[_iMuCltIdx].Clients[_i]].iReqId := Kanlink.MuClientListe[_iMuCltIdx].iReqId;
							Kanlink.ClientListe[Kanlink.MuClientListe[_iMuCltIdx].Clients[_i]].TimeOutLeft := Kanlink.MuClientListe[_iMuCltIdx].TimeOut;

							Kanlink.ServerData.HeaderV1Send[_i].Command := Kanlink.ClientListe[Kanlink.MuClientListe[_iMuCltIdx].Clients[_i]].Cmd;
							Kanlink.ServerData.HeaderV1Send[_i].CmdNr := Kanlink.ClientListe[Kanlink.MuClientListe[_iMuCltIdx].Clients[_i]].CmdOpt AND 16#00FF;

							Kanlink.ServerData.HeaderV1Send[_i].dataFormat := 5;
							Kanlink.ServerData.HeaderV1Send[_i].Length := UDINT_TO_UINT(Kanlink.ClientListe[Kanlink.MuClientListe[_iMuCltIdx].Clients[_i]].ReqLength);
							Kanlink.ServerData.HeaderV1Send[_i].ReqID := Kanlink.ClientListe[Kanlink.MuClientListe[_iMuCltIdx].Clients[_i]].iReqId;
							Kanlink.ServerData.HeaderV1Send[_i].Tag	:= _dCltIf.tag;

						END_IF

					END_FOR

					KLLib_SendData(ADR(Kanlink),0,0,ADR(Kanlink.MuClientListe[_iMuCltIdx].sClientAdr),-1,_iMuCltIdx,KLLIB_REQ);

					Kanlink.MuClientListe[_iMuCltIdx].xReqPending := TRUE;
					Kanlink.MuClientListe[_iMuCltIdx].iCycleWait := 0;

					FOR _i := 0 TO KLLIB_MAX_MUL DO

						IF (Kanlink.MuClientListe[_iMuCltIdx].Clients[_i] >= 0) THEN

							Kanlink.ClientListe[Kanlink.MuClientListe[_iMuCltIdx].Clients[_i]].xReqPending := TRUE;
							Kanlink.ClientListe[Kanlink.MuClientListe[_iMuCltIdx].Clients[_i]].iCycleWait := 0;
						END_IF

					END_FOR

					Kanlink._xSendClient := FALSE;

					RETURN;

				END_IF

			END_IF;

		END_IF;	// sendClient

#ifndef  HLKANLINK_AUTONOM  // wird MIT Framework gearbeitet
	ELSIF IFmnParam.Out.xParamOK AND IFmnEth.Out.xDataValid THEN

		Kanlink.ServerData.MetaInfoResp.KanLink_Hostname := IFmnEth.Out.IP.sHostname;
		Kanlink.ServerData.MetaInfoResp.Machine_type := WSTRING_TO_STRING(IFmnParam.Out.HeaderVersion.utfMachineType);
		Kanlink.ServerData.MetaInfoResp.DataModelTimeStamp := IFmnParam.Out.HeaderVersion.dtTimestamp;
		Kanlink.ServerData.MetaInfoResp.DataModelVersion := IFmnParam.Out.HeaderVersion.wVersion;

		Kanlink.ServerData.PingResp.KanLink_Hostname := IFmnEth.Out.IP.sHostname;

		_xInitOK := TRUE;

	END_IF
#else  // falls OHNE Framework gearbeitet wird
	ELSIF TRUE THEN
		_xInitOK := TRUE;
	END_IF
#endif

END_PROGRAM

PROGRAM _EXIT

	Kanlink.udp.close.enable	:= TRUE;
	Kanlink.udp.close.ident		:= Kanlink.udp.open.ident;
	Kanlink.udp.close;

END_PROGRAM
```

#### KanLinkInit.st - Initialization code
```iecst
(********************************************************************
 * COPYRIGHT -- Herbert Kannegiesser GmbH
 ********************************************************************
 * Program: KanLink
 * File: KanLinkInit.st
 * Author: stahlhut
 * Created: December 23, 2011
 ********************************************************************
 * Implementation of program KanLink
 ********************************************************************)

PROGRAM _INIT

	// Packet-Version auslesen mit MO_ver aus SYS_lib und für den Additional Status zur Verfügung stellen

	ST_name(0,ADR(_sName),0);
	ST_info(0,ADR(_state),ADR(_tcnr));

	_sPkgName := 'hlKanLink';

	IF ( MO_ver(ADR(_sPkgName), 0, ADR(_VerStruc)) = 0 ) THEN

		brsmemcpy(ADR(hlKanLinkStatAd.sPkgVersion), ADR(_VerStruc.version), SIZEOF(_VerStruc.version));

	ELSE

		hlKanLinkStatAd.sPkgVersion := '---';

	END_IF

	_xInitOK := FALSE;

	// nötige adressen initialisieren:
	Kanlink.adrSelf := ADR(Kanlink);
	Kanlink.CfgServer.adrKanlink := ADR(Kanlink);
	Kanlink.CfgClient.adrKanlink := ADR(Kanlink);

	FOR _i := 0 TO HLKANLINK_MAX_SERVERCONNS DO
		Kanlink.ServerListe[_i].adrInterface := ADR(IFhlKanLink.Server[_i]);
		KLLib_ReadServerPara(ADR(Kanlink.ServerListe[_i]), ADR( IFhlKanLink.Parameter.Server[_i]),ADR(Kanlink));
	END_FOR;

	FOR _i := 0 TO HLKANLINK_MAX_CLIENTCONNS DO
		KLLib_ReadClientPara(ADR(Kanlink.ClientListe[_i]),ADR(IFhlKanLink.Parameter.Client[_i]),ADR(Kanlink));
		Kanlink.ClientListe[_i].TimeOut := 140;
		Kanlink.ClientListe[_i].adrInterface := ADR(IFhlKanLink.Parameter.Client[_i]);
	END_FOR;

	// Create Log
	//****************************************************************************************************************
	// Log erzeugen
	//****************************************************************************************************************

	_kgArLogWrite.enable := TRUE;
	_kgArLogWrite.ident := 0;
	_kgArLogWrite.errornr := 50010;

	_AsArLogCreate(enable := TRUE, pName := ADR('hlKanLinkL'), len := 4096*1, memType := arlogUSRROM);

	IF _AsArLogCreate.status = ERR_OK THEN

		_kgArLogWrite.ident := _AsArLogCreate.ident;

	ELSIF _AsArLogCreate.status = arlogERR_EXISTING THEN

		_AsArLogGetInfo(enable := TRUE, pName := ADR('hlKanLinkL'));

		IF _AsArLogGetInfo.status = ERR_OK THEN

			_kgArLogWrite.ident := _AsArLogGetInfo.ident;

		END_IF

	END_IF

	//****************************************************************************************************************
	// Ringbuffer for Logs
	//****************************************************************************************************************

	_kgRBcreateKanLinklog(sName := '_klLogrb', bMemType := doUSRRAM, wCntEntry := 10, lLenEntry := SIZEOF(_LogEntry), wPtrWrite := _wPtrRBwrite, wPtrRead := _wPtrRBread, wPtrStart := _wPtrRBstart);

	IF _kgRBcreateKanLinklog.wStatus = ERR_OK THEN

		_wPtrRBloc := 0;

		_xRBReady := TRUE;

		_InsertRB.doIdent := _kgRBcreateKanLinklog.doIdent;
		_InsertRB.doLen := _kgRBcreateKanLinklog.doLen;
		_InsertRB.lLenEntry := SIZEOF(_LogEntry);
		_InsertRB.pEntry := ADR(_LogEntryIn);

		_ReadRB.doIdent := _kgRBcreateKanLinklog.doIdent;
		_ReadRB.doLen := _kgRBcreateKanLinklog.doLen;
		_ReadRB.lLenEntry := SIZEOF(_LogEntry);
		_ReadRB.pEntry := ADR(_LogEntry);

	ELSE

		_kgArLogWrite.logLevel := arlogLEVEL_INFO;
		_kgArLogWrite.text := 'Create Ringbuffer: {##AttrVar1}';
		_kgArLogWrite.var1 := _kgRBcreateKanLinklog.wStatus;
		_kgArLogWrite.var2 := 0;
		_kgArLogWrite();

	END_IF

	_wLogStep := 0;

	// Create StructureDescriptions
	//****************************************************************************************************************
	// Speicher allokoieren
	//****************************************************************************************************************

	_MemPartCreate(enable := TRUE, len := 8000);

	_LogEntryIn.wErrorNo := HLKANLINK_MSG_NO_STRUCDEF;

	IF _MemPartCreate.status = ERR_OK THEN

		_lTempMemIdent := _MemPartCreate.ident;

		_MemPartCreate(enable := TRUE, len := 8000);

		IF _MemPartCreate.status = ERR_OK THEN

			_lMemIdent := _MemPartCreate.ident;

			_MemAllocTemp(enable := TRUE, ident := _lTempMemIdent, len := 7500);

			IF _MemAllocTemp.status = ERR_OK THEN

				_lAdr := _MemAllocTemp.mem;
				_lLen := _MemAllocTemp.len;

				_wStatus := KLLib_CreateStrucDef(lPtrAdr := ADR(_lAdr), lPtrLen := ADR(_lLen), sRootName := 'hlKanLink:Kanlink.ServerData.MetaInfoResp', sItemName := '', lDataAdr := 0);

				IF _wStatus = ERR_OK THEN

					_MemAlloc(enable := TRUE, ident := _lMemIdent, len := _MemAllocTemp.len - _lLen);

					IF _MemAlloc.status = ERR_OK THEN

						_lPtrStrucDef[_HLKANLINK_IDX_STRUCDEF_RESP_0] := _MemAlloc.mem;
						_lPtrStrucLen[_HLKANLINK_IDX_STRUCDEF_RESP_0] := _MemAlloc.len;

						brsmemcpy(_MemAlloc.mem, _MemAllocTemp.mem, _MemAlloc.len);

						_MemFreeTemp(enable := TRUE, ident := _lTempMemIdent, mem := _MemAllocTemp.mem );

					ELSE

						_LogEntryIn.lAttr1 := _MemAlloc.status;
						_InsertRB(wPtrStart := _wPtrRBstart, wPtrRead := _wPtrRBread, wPtrWrite := _wPtrRBwrite);

					END_IF

				ELSE

					_LogEntryIn.lAttr1 := _wStatus;
					_InsertRB(wPtrStart := _wPtrRBstart, wPtrRead := _wPtrRBread, wPtrWrite := _wPtrRBwrite);

				END_IF

			ELSE

				_LogEntryIn.lAttr1 := _MemAllocTemp.status;
				_InsertRB(wPtrStart := _wPtrRBstart, wPtrRead := _wPtrRBread, wPtrWrite := _wPtrRBwrite);

			END_IF

		ELSE

			_LogEntryIn.lAttr1 := _MemPartCreate.status;
			_InsertRB(wPtrStart := _wPtrRBstart, wPtrRead := _wPtrRBread, wPtrWrite := _wPtrRBwrite);

		END_IF

	ELSE

		_LogEntryIn.lAttr1 := _MemPartCreate.status;
		_InsertRB(wPtrStart := _wPtrRBstart, wPtrRead := _wPtrRBread, wPtrWrite := _wPtrRBwrite);

	END_IF

END_PROGRAM
```

#### KL_SaveConfDO.st - Speichern der Parameter in Datenobjekt
```iecst
(********************************************************************
 * COPYRIGHT -- Herbert Kannegiesser GmbH
 ********************************************************************
 * Program: WetLink
 * File: WL_SaveConfDO.st
 * Author: stahlhut
 * Created: January 09, 2012
 ********************************************************************
 * Implementation of program WetLink
 ********************************************************************)

(* Speichern der Parameter in Datenobjekt *)
FUNCTION_BLOCK KL_SaveConfDO
CASE iSaveStep  OF
	0: ;
	 // DO vorhanden?

		status :=ERR_FUB_BUSY;

		DatObjInfo_0.enable := TRUE;
 		DatObjInfo_0.pName := adrName;
		DatObjInfo_0;
		IF DatObjInfo_0.status = ERR_FUB_BUSY THEN
  			// warten
		ELSIF DatObjInfo_0.status = 0 THEN
			// DO existiert, weiter mit löschen
			iSaveStep := 2;
		ELSIF DatObjInfo_0.status = doERR_MODULNOTFOUND THEN
			// Do existiert nicht, weiter mit Schreiben
			iSaveStep := 3;
		ELSE // fehler aufgetreten
			status := 3;
			iSaveStep := 0;
		END_IF;
	2: // löschen

		status :=ERR_FUB_BUSY;
		DatObjDelete_0(enable := 1 , ident := DatObjInfo_0.ident);
		CASE DatObjDelete_0.status OF
  			0: // fertig
				iSaveStep := 3;
			ERR_FUB_BUSY:
				// warten
			ELSE // fehler
				status :=4;
				iSaveStep := 0;
		END_CASE;
	3:
		DatObjCreate_0.enable := 1;
		DatObjCreate_0.MemType := doUSRROM;
		DatObjCreate_0.pName := adrName;
		DatObjCreate_0.pCpyData := adrDaten;
		DatObjCreate_0.len := len;
		DatObjCreate_0;
		CASE DatObjCreate_0.status OF
  			0: //fertig
				iSaveStep:= 0;
				status :=0;

			ERR_FUB_BUSY:
				// warten
				status := ERR_FUB_BUSY;
			ELSE
   				// fehler
				status := 5;
		END_CASE;
	ELSE
		iSaveStep := 0;
		status := 6;
END_CASE;

END_FUNCTION_BLOCK
```

#### KanLink.fun
```iecst
(********************************************************************
 * COPYRIGHT -- Herbert Kannegiesser GmbH
 ********************************************************************
 * Program: WetLink
 * File: WetLink.fun
 * Author: stahlhut
 * Created: January 09, 2012
 ********************************************************************
 * Functions and function blocks of program WetLink
 ********************************************************************)

FUNCTION_BLOCK KL_SaveConfDO (*Speichern der Parameter in Datenobjekt*)
	VAR_INPUT
		adrName : UDINT;
		adrDaten : UDINT;
		len : UDINT;
	END_VAR
	VAR_OUTPUT
		status : UINT;
		iSaveStep : INT;
		DatObjInfo_0 : DatObjInfo;
		DatObjDelete_0 : DatObjDelete;
		DatObjCreate_0 : DatObjCreate;
	END_VAR
END_FUNCTION_BLOCK
```

#### actGetServerReq.st
```iecst
(********************************************************************
 * COPYRIGHT --
 ********************************************************************
 * Program: hlKanLink
 * File: actGetServerReq.st
 * Author: stahlhut
 * Created: April 01, 2015
 ********************************************************************
 * Implementation of program hlKanLink
 ********************************************************************)

(* Kanlink Server/Request bearbeiten *)
ACTION actGetServerReq:

		Kanlink.MuServerListe.bMuServerIdx := 0;
		FOR _k := 0 TO KLLIB_MAX_MUL DO
			Kanlink.MuServerListe.Servers[_k] := -1;
			Kanlink.MuServerListe.MuServer[_k] := -1;
		END_FOR

		FOR _k := 0 TO KLLIB_MAX_MUL DO

			IF ((Kanlink.ServerData.HeaderV1Rec[_k].Command = 0) AND (Kanlink.ServerData.HeaderV1Rec[_k].ReqID = 0)) THEN
				EXIT;
			END_IF

			// Commandos unter 1000 sind für alle gleich:
			IF Kanlink.ServerData.HeaderV1Rec[_k].Command < 1000 THEN

				CASE Kanlink.ServerData.HeaderV1Rec[_k].Command OF
					0:   // MaschinenInfo Senden: Darf jeder lesen

						Kanlink.ServerData.HeaderV1Send[_k].Command := 1;
						Kanlink.ServerData.HeaderV1Send[_k].dataFormat := 5;
						Kanlink.ServerData.HeaderV1Send[_k].Length := 74;
						Kanlink.ServerData.HeaderV1Send[_k].Tag := Kanlink.ServerData.HeaderV1Rec[_k].Tag;
						Kanlink.ServerData.HeaderV1Send[_k].ReqID := Kanlink.ServerData.HeaderV1Rec[_k].ReqID;

						IF (Kanlink.ServerData.PreHeaderRec.HeaderVersion = 16#0101) THEN
							Kanlink.MuServerListe.Servers[_k]:= 32000;
							_sClientIPAdr := Kanlink.client_address;
						ELSE
							KLLib_SendData(ADR(Kanlink),ADR(Kanlink.ServerData.MetaInfoResp),74,ADR(Kanlink.client_address), -1,      -1,KLLIB_RESP);
							_iIdxFound := 32000;
						END_IF

					2:   // Response Ping: Darf jeder lesen

						Kanlink.ServerData.HeaderV1Send[_k].Command := 3;
						Kanlink.ServerData.HeaderV1Send[_k].dataFormat := 5;
						Kanlink.ServerData.HeaderV1Send[_k].Length := 17;
						Kanlink.ServerData.HeaderV1Send[_k].Tag := Kanlink.ServerData.HeaderV1Rec[_k].Tag;
						Kanlink.ServerData.HeaderV1Send[_k].ReqID := Kanlink.ServerData.HeaderV1Rec[_k].ReqID;

						IF (Kanlink.ServerData.PreHeaderRec.HeaderVersion = 16#0101) THEN
							Kanlink.MuServerListe.Servers[_k]:= 32000;
							_sClientIPAdr := Kanlink.client_address;
						ELSE
							KLLib_SendData(ADR(Kanlink),ADR(Kanlink.ServerData.PingResp),17,ADR(Kanlink.client_address), -1,      -1,KLLIB_RESP);
							_iIdxFound := 32000;
						END_IF

				END_CASE;

			ELSE
				// >= 1000 sind spezifische Daten

				// Anfrage Konfiguriert?
				// Zur Anfrage Verbindung raussuchen..
				_xIdxFound := FALSE;
				_iIdxFound := 32000;

				KL_BuildKey(Command := Kanlink.ServerData.HeaderV1Rec[_k].Command,CmdNr := UINT_TO_USINT( Kanlink.ServerData.HeaderV1Rec[_k].CmdNr AND 16#00FF) ,IPAdr := Kanlink.ServerData.IPAdr, adrKey:= ADR(Kanlink.RecKey));
				FOR _i := 0 TO HLKANLINK_MAX_SERVERCONNS  DO

					_ptrIndex ACCESS ADR(Kanlink.ServerListe[_i]);
					_dSrvIf ACCESS _ptrIndex.adrInterface;
					IF _ptrIndex.Adr = 0 THEN // wenn alle das Commando lesen dürfen/ Adresse und Area ausblenden
						IF Kanlink.RecKey.CmdKey = _ptrIndex.Key.CmdKey THEN // Index gefunden, beantworten:
							_xIdxFound := TRUE;
							_iIdxFound := _i;
							Kanlink.MuServerListe.Servers[_k] := _i;
							EXIT;
						END_IF;
					ELSE
						IF (Kanlink.RecKey.CmdKey = _ptrIndex.Key.CmdKey) AND (Kanlink.RecKey.IP_Key = _ptrIndex.Key.IP_Key) THEN // Index gefunden, beantworten:
							_xIdxFound := TRUE;
							_iIdxFound := _i;
							Kanlink.MuServerListe.Servers[_k]:= _i;
							EXIT;
						END_IF;
					END_IF;
				END_FOR

				IF (_k > 0) THEN
					FOR _i := 0 TO (_k - 1) DO
						IF (Kanlink.MuServerListe.Servers[_i] = Kanlink.MuServerListe.Servers[_k]) THEN
							Kanlink.MuServerListe.MuServer[_k] := USINT_TO_INT(Kanlink.MuServerListe.bMuServerIdx);
							Kanlink.MuServerListe.bMuServerIdx := Kanlink.MuServerListe.bMuServerIdx + 1;
							IF (Kanlink.MuServerListe.MuServer[_k] = 0) THEN
								Kanlink.MuServerListe.AdrRespData[Kanlink.MuServerListe.MuServer[_k]] := ADR(Kanlink.MuServerListe.RespData);
							ELSE
								Kanlink.MuServerListe.AdrRespData[Kanlink.MuServerListe.MuServer[_k]] := Kanlink.MuServerListe.AdrRespData[Kanlink.MuServerListe.MuServer[_k] - 1] + Kanlink.MuServerListe.lRespLength[Kanlink.MuServerListe.MuServer[_k] - 1];
							END_IF
							EXIT;
						END_IF
					END_FOR
				END_IF

				_xAdrErr := (_ptrIndex.AdrDataReq = 0) OR (_ptrIndex.AdrDataResp = 0);

				IF (_xIdxFound = FALSE) OR _xAdrErr THEN // Falls keine gültige Verbindung dann Fehlerframe senden
					// Fehlerframe senden:
					Kanlink.ServerData.HeaderV1Send[_k].Command := Kanlink.ServerData.HeaderV1Rec[_k].Command +1;
					Kanlink.ServerData.HeaderV1Send[_k].dataFormat := 255;
					Kanlink.ServerData.HeaderV1Send[_k].Length := 68;
					Kanlink.ServerData.HeaderV1Send[_k].Tag := Kanlink.ServerData.HeaderV1Rec[_k].Tag;
					Kanlink.ServerData.HeaderV1Send[_k].ReqID := Kanlink.ServerData.HeaderV1Rec[_k].ReqID;

					// Error Frame:
					Kanlink.ServerData.ErrorFrame.ErrorNumber := 2;
					strcpy(ADR(Kanlink.ServerData.ErrorFrame.ErrorText),ADR('request not supported'));

				ELSE
					// Empfangene Daten speichern:

					IF NOT( (_dSrvIf.iState <> 0) AND _ptrIndex.xReqManually) THEN  // falls Req bereits bearbeitet wird verwerfen
						_ptrIndex.iReqCnt := _ptrIndex.iReqCnt + 1;
						_dSrvIf.iState := 1;
						strcpy(ADR(_ptrIndex.sClientIPAdr),ADR(Kanlink.client_address));
						_sClientIPAdr := Kanlink.client_address;
						// todo längenüberprüfung _ptrIndex.ReqLength
						IF (_k = 0) THEN
							memcpy(_ptrIndex.AdrDataReq,ADR(Kanlink.ServerData.receive_data) + PreHeaderSize + HeaderSize,_ptrIndex.ReqLength);
						ELSE
							memcpy(_ptrIndex.AdrDataReq,ADR(Kanlink.ServerData.receive_data) + Kanlink.MuServerListe.wOffset[_k] + HeaderSize,_ptrIndex.ReqLength);
						END_IF

						_ptrIndex.iReqID := Kanlink.ServerData.HeaderV1Rec[_k].ReqID;
						_dSrvIf.out.tag	:= Kanlink.ServerData.HeaderV1Rec[_k].Tag;

						IF (_ptrIndex.CmdOpt AND KL_optOnReqCall) <> 0 THEN
							IF (Kanlink.MuServerListe.MuServer[_k] < 0) THEN
								KL_OnRecReq(adrReqData := _ptrIndex.AdrDataReq, adrRespData := _ptrIndex.AdrDataResp, adrKanlink := ADR(Kanlink),_ptrIndex.Cmd, adrUserData := IFhlKanLink.Parameter.adrUserTyp);
							ELSE
								KL_OnRecReq(adrReqData := _ptrIndex.AdrDataReq, adrRespData := Kanlink.MuServerListe.AdrRespData[Kanlink.MuServerListe.MuServer[_k]], adrKanlink := ADR(Kanlink),_ptrIndex.Cmd, adrUserData := IFhlKanLink.Parameter.adrUserTyp);
								Kanlink.MuServerListe.lRespLength[Kanlink.MuServerListe.MuServer[_k]] := _ptrIndex.RespLength;
							END_IF
						END_IF;
						IF _ptrIndex.xReqManually = 0 THEN

							Kanlink.ServerData.HeaderV1Send[_k].Command := _ptrIndex.Cmd + 1;
							Kanlink.ServerData.HeaderV1Send[_k].dataFormat := 5;
							Kanlink.ServerData.HeaderV1Send[_k].Length := UDINT_TO_UINT( _ptrIndex.RespLength);
							Kanlink.ServerData.HeaderV1Send[_k].ReqID := _ptrIndex.iReqID;
							Kanlink.ServerData.HeaderV1Send[_k].CmdNr := _ptrIndex.CmdOpt AND 16#00FF;
							Kanlink.ServerData.HeaderV1Send[_k].Tag	:= _dSrvIf.tag;
							_ptrIndex.iConnectionTimer := 0;
						END_IF;
					END_IF;

				END_IF;

			END_IF;

		END_FOR

		IF (Kanlink.ServerData.PreHeaderRec.HeaderVersion = 16#0101) THEN
			KLLib_SendData(ADR(Kanlink),0,0,ADR(_sClientIPAdr),-1,0,KLLIB_RESP);
		ELSIF (_iIdxFound <> 32000) THEN
			KLLib_SendData(ADR(Kanlink),_ptrIndex.AdrDataResp,_ptrIndex.RespLength,ADR(_ptrIndex.sClientIPAdr), -1,      -1,KLLIB_RESP);
		END_IF

END_ACTION
```

#### actResponse.st
```iecst
(********************************************************************
 * COPYRIGHT --
 ********************************************************************
 * Program: hlKanLink
 * File: actResponse.st
 * Author: stahlhut
 * Created: April 01, 2015
 ********************************************************************
 * Implementation of program hlKanLink
 ********************************************************************)

(* Response eines Servers bearbeiten *)
ACTION actResponse:

		FOR _k := 0 TO KLLIB_MAX_MUL DO
			Kanlink.MuServerListe.Servers[_k] := -1;
		END_FOR

		FOR _k := 0 TO KLLIB_MAX_MUL DO

			IF ((Kanlink.ServerData.HeaderV1Rec[_k].Command = 0) AND (Kanlink.ServerData.HeaderV1Rec[_k].ReqID = 0)) THEN
				EXIT;
			END_IF

			KL_BuildKey(Command := Kanlink.ServerData.HeaderV1Rec[_k].Command,CmdNr := UINT_TO_USINT( Kanlink.ServerData.HeaderV1Rec[_k].CmdNr AND 16#00FF) ,IPAdr := Kanlink.ServerData.IPAdr, adrKey:= ADR(Kanlink.RecKey));

			_xIdxFound := FALSE;
			FOR _i := 0 TO HLKANLINK_MAX_CLIENTCONNS DO
				_dClient ACCESS ADR(Kanlink.ClientListe[_i]);

				IF (Kanlink.RecKey.CmdKey = _dClient.Key.CmdKey) AND (Kanlink.RecKey.IP_Key = _dClient.Key.IP_Key) THEN // Index gefunden, beantworten:
					_xIdxFound := TRUE;
					Kanlink.MuServerListe.Servers[_k] := _i;
					EXIT;
				END_IF;
			END_FOR

			_xAdrOK := _dClient.AdrDataResp <> 0 ;

			IF _xIdxFound AND _xAdrOK THEN
				_dClient.xReqPending := FALSE;
				IF (_dClient.MuClient >= 0) THEN
					IF (Kanlink.ServerData.PreHeaderRec.HeaderVersion = 16#0101) THEN
						IF (Kanlink.MuClientListe[_dClient.MuClient].bUse = 2) THEN
							Kanlink.MuClientListe[_dClient.MuClient].bUse := 1;
						END_IF
					ELSIF (Kanlink.ServerData.PreHeaderRec.HeaderVersion = 16#0100) THEN
						Kanlink.MuClientListe[_dClient.MuClient].bUse := 255;
					END_IF
					IF ((Kanlink.MuClientListe[_dClient.MuClient].bUse <> 0) AND (Kanlink.MuClientListe[_dClient.MuClient].bUse <> 255)) THEN
						Kanlink.MuClientListe[_dClient.MuClient].xReqPending := FALSE;
					END_IF
				END_IF

				IF _dClient.iTimeOutCnt > 0 THEN
					_dClient.iTimeOutCnt := _dClient.iTimeOutCnt - 1;
				END_IF;
				IF _dClient.adrInterface <> 0 THEN
					_dCltIf ACCESS _dClient.adrInterface;
					_dCltIf.iState := 3;
				END_IF;

				IF (_k = 0) THEN
					memcpy(_dClient.AdrDataResp,ADR(Kanlink.ServerData.receive_data) + PreHeaderSize + HeaderSize,_dClient.RespLength);
				ELSE
					memcpy(_dClient.AdrDataResp,ADR(Kanlink.ServerData.receive_data) + Kanlink.MuServerListe.wOffset[_k] + HeaderSize,_dClient.RespLength);
				END_IF

				_dCltIf.out.recTag := Kanlink.ServerData.HeaderV1Rec[_k].Tag;

		  	END_IF;

		END_FOR

		_iCltRespCnt := _iCltRespCnt + 1;
		Kanlink._xGetClientResp := FALSE;

		Kanlink._xSendClient := TRUE; // Daten einsortiert, nix weiter zutun also Clients bearbeiten
		Kanlink.udp.rec.enable := 1;

END_ACTION
```

### Library Logical/Standard/Kanlink/KGFramework/Pkg_hlKanLink/KanLinkLib (IEC, version 0.94.5) - KanlinkHilfsfunktionen
Depends on: AsUDP, asstring, AsARCfg, brsystem, sys_lib, AsArLog, AsIODiag, AsETH, DataObj, KL_UserLib, KGstdLib

#### CmdBTxfer.typ - Commando Batch Transfer
```iecst
(********************************************************************
 * COPYRIGHT -- Herbert Kannegiesser GmbH
 ********************************************************************
 * Library: Kanlink Commando 1000 BatchTransfer
 * File:
 * Author: stahlhut
 * Created: 20.03.2012
 ********************************************************************
 * Data types of library WetLinkLib
 ********************************************************************)
(*Interne Strukturen*)

TYPE
	KL_BTxf_typ : 	STRUCT  (*Batch Transfer Server*)
		Req : KLreq1000_BTH_typ;
		Resp : KLresp1000_BTH_typ;
	END_STRUCT;
	KLreq1000_BTH_typ : 	STRUCT
		xHready : BOOL;
		xHreadyForLoad : BOOL;
		xHbatchReceived : BOOL;
		xHtransferzoneOccupied : BOOL;
		xHreqCtrlTransfer : BOOL;
		xHtransferRunning : BOOL;
		xHwaitingForTransfer : BOOL;
		xHshiftBatches : BOOL;
		wHstate : UINT;
		bHcmdAutomatic : USINT;
		xHreserve : ARRAY[1..5]OF BOOL;
		wTimeToReadyForLoad : UINT;
		wRemainProctime : UINT; (*Remaining Processtime / Verbleibende Prozesszeit*)
	END_STRUCT;
	KLresp1000_BTH_typ : 	STRUCT
		xHsCmdFinishProcess : BOOL;
		xHsReqForUnload : BOOL;
		xHsUnloading : BOOL;
		xHsReqCtrlTransfer : BOOL;
		xHsTransferRunning : BOOL;
		xHsRes : BOOL;
		wState : UINT;
		bCmdAuto : USINT;
		xCmdStartProcess : BOOL;
		xHsDataValid : BOOL;
		xHsRes2 : ARRAY[0..2]OF BOOL;
		wCntLoads : UINT;
		BatchData : BatchData_typ;
	END_STRUCT;
END_TYPE
```

#### CmdBI.typ - BatchInformation / 1002
```iecst
(********************************************************************
 * COPYRIGHT -- Herbert Kannegiesser GmbH
 ********************************************************************
 * Library: Kanlink Cmd 1002 Batch Information
 * File: WetLinkLib.typ
 * Author: stahlhut
 * Created: 20.03.2012
 ********************************************************************
 * Data types of library Kanlink
 ********************************************************************)
(*Kommando*)

TYPE
	KLreq1002_Info_typ : 	STRUCT
		wCntPositions : UINT;
		wNoOfPosition : ARRAY[0..5]OF UINT;
		wRes : UINT;
	END_STRUCT;
	KLresp1002_Info_typ : 	STRUCT
		wCntPositions : UINT;
		wNoOfPositions : ARRAY[0..5]OF UINT;
		wRes : UINT;
		BatchData : ARRAY[0..5]OF BatchData_typ;
	END_STRUCT;
	KL_BI_typ : 	STRUCT
		Req : KLreq1002_Info_typ;
		Resp : KLresp1002_Info_typ;
	END_STRUCT;
END_TYPE
```
